LIN {X 0,Y 567.172,Z 389.799,A -85,B 0,C 180,E1 24706.932,E2 24706.932} C_VEL
LIN {X 0,Y 570.884,Z 340.567,A -85,B 0,C 180,E1 24705.981,E2 24705.981} C_VEL
LIN {X 0,Y 571.881,Z 338.159,A -85,B 0,C 180,E1 24705.833,E2 24705.833} C_VEL
LIN {X 0,Y 579.094,Z 319.344,A -85,B 0,C 180,E1 24704.229,E2 24704.229} C_VEL
LIN {X 0,Y 582.937,Z 311.16,A -85,B 0,C 180,E1 24703.458,E2 24703.458} C_VEL
LIN {X 0,Y 582.832,Z 309.162,A -85,B 0,C 180,E1 24702.394,E2 24702.394} C_VEL
LIN {X 0,Y 582.89,Z 308.585,A -85,B 0,C 180,E1 24701.727,E2 24701.727} C_VEL
LIN {X 0,Y 582.338,Z 310.355,A -85,B 0,C 180,E1 24700.405,E2 24700.405} C_VEL
LIN {X 0,Y 574.337,Z 326.452,A -85,B 0,C 180,E1 24698.682,E2 24698.682} C_VEL
LIN {X 0,Y 566.735,Z 346.819,A -85,B 0,C 180,E1 24696.671,E2 24696.671} C_VEL
LIN {X 0,Y 559.494,Z 373.809,A -85,B 0,C 180,E1 24694.198,E2 24694.198} C_VEL
LIN {X 0,Y 554.301,Z 400.115,A -85,B 0,C 180,E1 24691.96,E2 24691.96} C_VEL
LIN {X 0,Y 555.519,Z 423.333,A -85,B 0,C 180,E1 24690.693,E2 24690.693} C_VEL
LIN {X 0,Y 556.922,Z 451.305,A -85,B 0,C 180,E1 24689.365,E2 24689.365} C_VEL
LIN {X 0,Y 558.184,Z 484.283,A -85,B 0,C 180,E1 24688.02,E2 24688.02} C_VEL
LIN {X 0,Y 558.47,Z 501.799,A -85,B 0,C 180,E1 24687.4,E2 24687.4} C_VEL
LIN {X 0,Y 549.884,Z 603.402,A -85,B 0,C 180,E1 24685.067,E2 24685.067} C_VEL
LIN {X 0,Y 544.198,Z 689.935,A -85,B 0,C 180,E1 24683.104,E2 24683.104} C_VEL
LIN {X 0,Y 542.555,Z 713.994,A -85,B 0,C 180,E1 24682.34,E2 24682.34} C_VEL
LIN {X 0,Y 541.005,Z 736.005,A -85,B 0,C 180,E1 24681.432,E2 24681.432} C_VEL
LIN {X 0,Y 539.398,Z 756.989,A -85,B 0,C 180,E1 24680.339,E2 24680.339} C_VEL
LIN {X 0,Y 538.011,Z 774.87,A -85,B 0,C 180,E1 24679.205,E2 24679.205} C_VEL
LIN {X 0,Y 536.611,Z 791.893,A -85,B 0,C 180,E1 24677.906,E2 24677.906} C_VEL
LIN {X 0,Y 535.34,Z 806.843,A -85,B 0,C 180,E1 24676.549,E2 24676.549} C_VEL
LIN {X 0,Y 534.145,Z 820.367,A -85,B 0,C 180,E1 24675.082,E2 24675.082} C_VEL
LIN {X 0,Y 533.023,Z 832.916,A -85,B 0,C 180,E1 24673.451,E2 24673.451} C_VEL
LIN {X 0,Y 532.018,Z 843.847,A -85,B 0,C 180,E1 24671.711,E2 24671.711} C_VEL
LIN {X 0,Y 531.163,Z 853.18,A -85,B 0,C 180,E1 24669.864,E2 24669.864} C_VEL
LIN {X 0,Y 530.507,Z 860.457,A -85,B 0,C 180,E1 24668.017,E2 24668.017} C_VEL
LIN {X 0,Y 530,Z 866.128,A -85,B 0,C 180,E1 24666.065,E2 24666.065} C_VEL
LIN {X 0,Y 529.624,Z 869.937,A -85,B 0,C 180,E1 24664.114,E2 24664.114} C_VEL
LIN {X 0,Y 529.372,Z 871.943,A -85,B 0,C 180,E1 24662.165,E2 24662.165} C_VEL
LIN {X 0,Y 529.209,Z 872.179,A -85,B 0,C 180,E1 24660.108,E2 24660.108} C_VEL
LIN {X 0,Y 529.126,Z 870.512,A -85,B 0,C 180,E1 24658.051,E2 24658.051} C_VEL
LIN {X 0,Y 529.146,Z 867.199,A -85,B 0,C 180,E1 24656.099,E2 24656.099} C_VEL
LIN {X 0,Y 529.276,Z 862.125,A -85,B 0,C 180,E1 24654.145,E2 24654.145} C_VEL
LIN {X 0,Y 529.52,Z 855.186,A -85,B 0,C 180,E1 24652.186,E2 24652.186} C_VEL
LIN {X 0,Y 529.941,Z 846.185,A -85,B 0,C 180,E1 24650.223,E2 24650.223} C_VEL
LIN {X 0,Y 530.543,Z 835.567,A -85,B 0,C 180,E1 24648.366,E2 24648.366} C_VEL
LIN {X 0,Y 531.311,Z 823.375,A -85,B 0,C 180,E1 24646.616,E2 24646.616} C_VEL
LIN {X 0,Y 532.271,Z 809.122,A -85,B 0,C 180,E1 24644.921,E2 24644.921} C_VEL
LIN {X 0,Y 533.351,Z 793.597,A -85,B 0,C 180,E1 24643.387,E2 24643.387} C_VEL
LIN {X 0,Y 534.503,Z 776.998,A -85,B 0,C 180,E1 24642.021,E2 24642.021} C_VEL
LIN {X 0,Y 535.659,Z 759.422,A -85,B 0,C 180,E1 24640.82,E2 24640.82} C_VEL
LIN {X 0,Y 536.845,Z 740.956,A -85,B 0,C 180,E1 24639.788,E2 24639.788} C_VEL
LIN {X 0,Y 537.985,Z 720.972,A -85,B 0,C 180,E1 24638.894,E2 24638.894} C_VEL
LIN {X 0,Y 538.984,Z 700.182,A -85,B 0,C 180,E1 24638.188,E2 24638.188} C_VEL
LIN {X 0,Y 539.819,Z 679.295,A -85,B 0,C 180,E1 24637.684,E2 24637.684} C_VEL
LIN {X 0,Y 545.343,Z 494.327,A -85,B 0,C 180,E1 24634.546,E2 24634.546} C_VEL
LIN {X 0,Y 540.838,Z 450.424,A -85,B 0,C 180,E1 24633.456,E2 24633.456} C_VEL
LIN {X 0,Y 544.277,Z 398.054,A -85,B 0,C 180,E1 24629.86,E2 24629.86} C_VEL
LIN {X 0,Y 547.874,Z 348.579,A -85,B 0,C 180,E1 24626.428,E2 24626.428} C_VEL
LIN {X 0,Y 552.064,Z 296.542,A -85,B 0,C 180,E1 24622.776,E2 24622.776} C_VEL
LIN {X 0,Y 553.399,Z 279.163,A -85,B 0,C 180,E1 24621.532,E2 24621.532} C_VEL
LIN {X 0,Y 544.537,Z 255.5,A -85,B 0,C 180,E1 24618.998,E2 24618.998} C_VEL
LIN {X 0,Y 535.075,Z 232.411,A -85,B 0,C 180,E1 24616.318,E2 24616.318} C_VEL
LIN {X 0,Y 534.781,Z 231.7,A -85,B 0,C 180,E1 24616.227,E2 24616.227} C_VEL
LIN {X 0,Y 536.691,Z 232.864,A -85,B 0,C 180,E1 24615.941,E2 24615.941} C_VEL
LIN {X 0,Y 546.06,Z 252.219,A -85,B 0,C 180,E1 24613.597,E2 24613.597} C_VEL
LIN {X 0,Y 554.586,Z 272.537,A -85,B 0,C 180,E1 24611.251,E2 24611.251} C_VEL
LIN {X 0,Y 561.348,Z 291.078,A -85,B 0,C 180,E1 24609.21,E2 24609.21} C_VEL
LIN {X 0,Y 561.17,Z 298.745,A -85,B 0,C 180,E1 24608.658,E2 24608.658} C_VEL
LIN {X 0,Y 560.235,Z 305.401,A -85,B 0,C 180,E1 24608.261,E2 24608.261} C_VEL
LIN {X 0,Y 555.035,Z 324.312,A -85,B 0,C 180,E1 24607.416,E2 24607.416} C_VEL
LIN {X 0,Y 554.398,Z 330.093,A -85,B 0,C 180,E1 24607.081,E2 24607.081} C_VEL
LIN {X 0,Y 554.416,Z 348.963,A -85,B 0,C 180,E1 24605.852,E2 24605.852} C_VEL
LIN {X 0,Y 552.164,Z 359.982,A -85,B 0,C 180,E1 24605.442,E2 24605.442} C_VEL
LIN {X 0,Y 549.54,Z 449.417,A -85,B 0,C 180,E1 24604.138,E2 24604.138} C_VEL
LIN {X 0,Y 546.257,Z 527.382,A -85,B 0,C 180,E1 24602.815,E2 24602.815} C_VEL
LIN {X 0,Y 541.758,Z 616.567,A -85,B 0,C 180,E1 24601.087,E2 24601.087} C_VEL
LIN {X 0,Y 540.542,Z 646.224,A -85,B 0,C 180,E1 24600.4,E2 24600.4} C_VEL
LIN {X 0,Y 539.38,Z 668.071,A -85,B 0,C 180,E1 24599.698,E2 24599.698} C_VEL
LIN {X 0,Y 537.858,Z 689.945,A -85,B 0,C 180,E1 24598.783,E2 24598.783} C_VEL
LIN {X 0,Y 536.147,Z 710.107,A -85,B 0,C 180,E1 24597.73,E2 24597.73} C_VEL
LIN {X 0,Y 534.288,Z 729.488,A -85,B 0,C 180,E1 24596.509,E2 24596.509} C_VEL
LIN {X 0,Y 532.25,Z 748.721,A -85,B 0,C 180,E1 24595.064,E2 24595.064} C_VEL
LIN {X 0,Y 530.139,Z 767.337,A -85,B 0,C 180,E1 24593.403,E2 24593.403} C_VEL
LIN {X 0,Y 528.194,Z 784.001,A -85,B 0,C 180,E1 24591.645,E2 24591.645} C_VEL
LIN {X 0,Y 526.509,Z 798.406,A -85,B 0,C 180,E1 24589.873,E2 24589.873} C_VEL
LIN {X 0,Y 524.913,Z 812.343,A -85,B 0,C 180,E1 24587.86,E2 24587.86} C_VEL
LIN {X 0,Y 523.561,Z 824.713,A -85,B 0,C 180,E1 24585.732,E2 24585.732} C_VEL
LIN {X 0,Y 522.516,Z 835.264,A -85,B 0,C 180,E1 24583.562,E2 24583.562} C_VEL
LIN {X 0,Y 521.742,Z 844.408,A -85,B 0,C 180,E1 24581.273,E2 24581.273} C_VEL
LIN {X 0,Y 521.227,Z 851.534,A -85,B 0,C 180,E1 24579.051,E2 24579.051} C_VEL
LIN {X 0,Y 520.916,Z 857.237,A -85,B 0,C 180,E1 24576.724,E2 24576.724} C_VEL
LIN {X 0,Y 520.738,Z 861.151,A -85,B 0,C 180,E1 24574.405,E2 24574.405} C_VEL
LIN {X 0,Y 520.657,Z 863.456,A -85,B 0,C 180,E1 24572.091,E2 24572.091} C_VEL
LIN {X 0,Y 520.639,Z 864.185,A -85,B 0,C 180,E1 24569.78,E2 24569.78} C_VEL
LIN {X 0,Y 520.658,Z 863.243,A -85,B 0,C 180,E1 24567.468,E2 24567.468} C_VEL
LIN {X 0,Y 520.758,Z 860.648,A -85,B 0,C 180,E1 24565.154,E2 24565.154} C_VEL
LIN {X 0,Y 520.942,Z 856.196,A -85,B 0,C 180,E1 24562.722,E2 24562.722} C_VEL
LIN {X 0,Y 521.293,Z 850.544,A -85,B 0,C 180,E1 24560.505,E2 24560.505} C_VEL
LIN {X 0,Y 521.889,Z 842.757,A -85,B 0,C 180,E1 24558.17,E2 24558.17} C_VEL
LIN {X 0,Y 522.691,Z 833.442,A -85,B 0,C 180,E1 24555.94,E2 24555.94} C_VEL
LIN {X 0,Y 523.79,Z 822.558,A -85,B 0,C 180,E1 24553.783,E2 24553.783} C_VEL
LIN {X 0,Y 525.167,Z 809.983,A -85,B 0,C 180,E1 24551.69,E2 24551.69} C_VEL
LIN {X 0,Y 526.732,Z 796.54,A -85,B 0,C 180,E1 24549.788,E2 24549.788} C_VEL
LIN {X 0,Y 528.506,Z 781.567,A -85,B 0,C 180,E1 24547.979,E2 24547.979} C_VEL
LIN {X 0,Y 530.475,Z 764.694,A -85,B 0,C 180,E1 24546.247,E2 24546.247} C_VEL
LIN {X 0,Y 532.444,Z 747.087,A -85,B 0,C 180,E1 24544.708,E2 24544.708} C_VEL
LIN {X 0,Y 534.424,Z 728.325,A -85,B 0,C 180,E1 24543.318,E2 24543.318} C_VEL
LIN {X 0,Y 536.282,Z 708.692,A -85,B 0,C 180,E1 24542.096,E2 24542.096} C_VEL
LIN {X 0,Y 537.972,Z 688.594,A -85,B 0,C 180,E1 24541.062,E2 24541.062} C_VEL
LIN {X 0,Y 539.445,Z 667.47,A -85,B 0,C 180,E1 24540.185,E2 24540.185} C_VEL
LIN {X 0,Y 540.613,Z 645.234,A -85,B 0,C 180,E1 24539.477,E2 24539.477} C_VEL
LIN {X 0,Y 541.962,Z 612.731,A -85,B 0,C 180,E1 24538.738,E2 24538.738} C_VEL
LIN {X 0,Y 546.474,Z 523.52,A -85,B 0,C 180,E1 24537.02,E2 24537.02} C_VEL
LIN {X 0,Y 549.681,Z 446.416,A -85,B 0,C 180,E1 24535.721,E2 24535.721} C_VEL
LIN {X 0,Y 552.294,Z 358.711,A -85,B 0,C 180,E1 24534.437,E2 24534.437} C_VEL
LIN {X 0,Y 554.559,Z 348.099,A -85,B 0,C 180,E1 24534,E2 24534} C_VEL
LIN {X 0,Y 554.663,Z 312.521,A -85,B 0,C 180,E1 24531.609,E2 24531.609} C_VEL
LIN {X 0,Y 554.973,Z 294.272,A -85,B 0,C 180,E1 24530.293,E2 24530.293} C_VEL
LIN {X 0,Y 547.767,Z 275.074,A -85,B 0,C 180,E1 24528.139,E2 24528.139} C_VEL
LIN {X 0,Y 539.853,Z 256.334,A -85,B 0,C 180,E1 24525.942,E2 24525.942} C_VEL
LIN {X 0,Y 532.349,Z 240.84,A -85,B 0,C 180,E1 24524.024,E2 24524.024} C_VEL
LIN {X 0,Y 526.336,Z 229.281,A -85,B 0,C 180,E1 24522.555,E2 24522.555} C_VEL
LIN {X 0,Y 523.694,Z 224.562,A -85,B 0,C 180,E1 24521.933,E2 24521.933} C_VEL
LIN {X 0,Y 521.964,Z 221.334,A -85,B 0,C 180,E1 24521.515,E2 24521.515} C_VEL
LIN {X 0,Y 521.744,Z 220.235,A -85,B 0,C 180,E1 24521.39,E2 24521.39} C_VEL
LIN {X 0,Y 521.743,Z 220.233,A -85,B 0,C 180,E1 24517.965,E2 24517.965} C_VEL
LIN {X 0,Y 521.737,Z 220.239,A -85,B 0,C 180,E1 24514.505,E2 24514.505} C_VEL
LIN {X 0,Y 521.735,Z 220.239,A -85,B 0,C 180,E1 24511.033,E2 24511.033} C_VEL
LIN {X 0,Y 521.739,Z 220.219,A -85,B 0,C 180,E1 24507.632,E2 24507.632} C_VEL
LIN {X 0,Y 521.742,Z 220.211,A -85,B 0,C 180,E1 24504.185,E2 24504.185} C_VEL
LIN {X 0,Y 521.737,Z 220.238,A -85,B 0,C 180,E1 24500.734,E2 24500.734} C_VEL
LIN {X 0,Y 521.741,Z 220.21,A -85,B 0,C 180,E1 24497.281,E2 24497.281} C_VEL
LIN {X 0,Y 521.732,Z 220.223,A -85,B 0,C 180,E1 24493.861,E2 24493.861} C_VEL
LIN {X 0,Y 521.742,Z 220.225,A -85,B 0,C 180,E1 24490.378,E2 24490.378} C_VEL
LIN {X 0,Y 521.745,Z 220.21,A -85,B 0,C 180,E1 24486.922,E2 24486.922} C_VEL
LIN {X 0,Y 521.729,Z 220.239,A -85,B 0,C 180,E1 24483.406,E2 24483.406} C_VEL
LIN {X 0,Y 521.726,Z 220.202,A -85,B 0,C 180,E1 24479.89,E2 24479.89} C_VEL
LIN {X 0,Y 521.744,Z 220.238,A -85,B 0,C 180,E1 24476.484,E2 24476.484} C_VEL
LIN {X 0,Y 521.744,Z 220.198,A -85,B 0,C 180,E1 24472.955,E2 24472.955} C_VEL
LIN {X 0,Y 521.72,Z 220.241,A -85,B 0,C 180,E1 24469.476,E2 24469.476} C_VEL
LIN {X 0,Y 521.739,Z 220.242,A -85,B 0,C 180,E1 24466.026,E2 24466.026} C_VEL
LIN {X 0,Y 521.749,Z 220.241,A -85,B 0,C 180,E1 24462.605,E2 24462.605} C_VEL
LIN {X 0,Y 521.717,Z 220.239,A -85,B 0,C 180,E1 24459.233,E2 24459.233} C_VEL
LIN {X 0,Y 521.722,Z 220.235,A -85,B 0,C 180,E1 24455.787,E2 24455.787} C_VEL
LIN {X 0,Y 521.753,Z 220.235,A -85,B 0,C 180,E1 24452.369,E2 24452.369} C_VEL
LIN {X 0,Y 521.722,Z 220.239,A -85,B 0,C 180,E1 24448.946,E2 24448.946} C_VEL
LIN {X 0,Y 521.754,Z 220.325,A -85,B 0,C 180,E1 24446.612,E2 24446.612} C_VEL
LIN {X 0,Y 522.874,Z 223.439,A -85,B 0,C 180,E1 24446.187,E2 24446.187} C_VEL
LIN {X 0,Y 524.045,Z 225.27,A -85,B 0,C 180,E1 24445.878,E2 24445.878} C_VEL
LIN {X 0,Y 525.794,Z 228.852,A -85,B 0,C 180,E1 24445.347,E2 24445.347} C_VEL
LIN {X 0,Y 533.823,Z 244.524,A -85,B 0,C 180,E1 24443.04,E2 24443.04} C_VEL
LIN {X 0,Y 543.759,Z 264.219,A -85,B 0,C 180,E1 24440.351,E2 24440.351} C_VEL
LIN {X 0,Y 556.286,Z 289.963,A -85,B 0,C 180,E1 24437.168,E2 24437.168} C_VEL
LIN {X 0,Y 561.303,Z 300.628,A -85,B 0,C 180,E1 24435.946,E2 24435.946} C_VEL
LIN {X 0,Y 559.967,Z 313.808,A -85,B 0,C 180,E1 24435.173,E2 24435.173} C_VEL
LIN {X 0,Y 562.81,Z 340.382,A -85,B 0,C 180,E1 24434.457,E2 24434.457} C_VEL
LIN {X 0,Y 554.944,Z 572.433,A -85,B 0,C 180,E1 24430.918,E2 24430.918} C_VEL
LIN {X 0,Y 551.384,Z 692.781,A -85,B 0,C 180,E1 24429.119,E2 24429.119} C_VEL
LIN {X 0,Y 549.935,Z 717.309,A -85,B 0,C 180,E1 24428.579,E2 24428.579} C_VEL
LIN {X 0,Y 548.22,Z 740.807,A -85,B 0,C 180,E1 24427.893,E2 24427.893} C_VEL
LIN {X 0,Y 546.127,Z 763.625,A -85,B 0,C 180,E1 24427.035,E2 24427.035} C_VEL
LIN {X 0,Y 543.758,Z 786.648,A -85,B 0,C 180,E1 24425.992,E2 24425.992} C_VEL
LIN {X 0,Y 541.136,Z 809.081,A -85,B 0,C 180,E1 24424.753,E2 24424.753} C_VEL
LIN {X 0,Y 538.432,Z 830.883,A -85,B 0,C 180,E1 24423.345,E2 24423.345} C_VEL
LIN {X 0,Y 535.859,Z 850.246,A -85,B 0,C 180,E1 24421.875,E2 24421.875} C_VEL
LIN {X 0,Y 533.106,Z 870.475,A -85,B 0,C 180,E1 24420.114,E2 24420.114} C_VEL
LIN {X 0,Y 530.656,Z 888,A -85,B 0,C 180,E1 24418.348,E2 24418.348} C_VEL
LIN {X 0,Y 528.37,Z 904.978,A -85,B 0,C 180,E1 24416.405,E2 24416.405} C_VEL
LIN {X 0,Y 526.295,Z 920.525,A -85,B 0,C 180,E1 24414.348,E2 24414.348} C_VEL
LIN {X 0,Y 524.481,Z 935.456,A -85,B 0,C 180,E1 24412.099,E2 24412.099} C_VEL
LIN {X 0,Y 523.037,Z 948.215,A -85,B 0,C 180,E1 24409.854,E2 24409.854} C_VEL
LIN {X 0,Y 521.869,Z 960.375,A -85,B 0,C 180,E1 24407.391,E2 24407.391} C_VEL
LIN {X 0,Y 521.085,Z 970.191,A -85,B 0,C 180,E1 24405.013,E2 24405.013} C_VEL
LIN {X 0,Y 520.553,Z 978.856,A -85,B 0,C 180,E1 24402.536,E2 24402.536} C_VEL
LIN {X 0,Y 520.257,Z 985.967,A -85,B 0,C 180,E1 24399.961,E2 24399.961} C_VEL
LIN {X 0,Y 520.116,Z 990.812,A -85,B 0,C 180,E1 24397.734,E2 24397.734} C_VEL
LIN {X 0,Y 520.085,Z 994.867,A -85,B 0,C 180,E1 24395.184,E2 24395.184} C_VEL
LIN {X 0,Y 520.101,Z 997.064,A -85,B 0,C 180,E1 24392.865,E2 24392.865} C_VEL
LIN {X 0,Y 520.12,Z 997.946,A -85,B 0,C 180,E1 24390.771,E2 24390.771} C_VEL
LIN {X 0,Y 520.139,Z 997.696,A -85,B 0,C 180,E1 24388.439,E2 24388.439} C_VEL
LIN {X 0,Y 520.139,Z 995.709,A -85,B 0,C 180,E1 24385.811,E2 24385.811} C_VEL
LIN {X 0,Y 520.149,Z 992.525,A -85,B 0,C 180,E1 24383.488,E2 24383.488} C_VEL
LIN {X 0,Y 520.233,Z 987.22,A -85,B 0,C 180,E1 24380.82,E2 24380.82} C_VEL
LIN {X 0,Y 520.439,Z 980.92,A -85,B 0,C 180,E1 24378.474,E2 24378.474} C_VEL
LIN {X 0,Y 520.81,Z 973.556,A -85,B 0,C 180,E1 24376.228,E2 24376.228} C_VEL
LIN {X 0,Y 521.5,Z 963.155,A -85,B 0,C 180,E1 24373.629,E2 24373.629} C_VEL
LIN {X 0,Y 522.274,Z 953.521,A -85,B 0,C 180,E1 24371.585,E2 24371.585} C_VEL
LIN {X 0,Y 523.524,Z 940.476,A -85,B 0,C 180,E1 24369.191,E2 24369.191} C_VEL
LIN {X 0,Y 524.882,Z 927.409,A -85,B 0,C 180,E1 24367.131,E2 24367.131} C_VEL
LIN {X 0,Y 526.69,Z 911.753,A -85,B 0,C 180,E1 24364.953,E2 24364.953} C_VEL
LIN {X 0,Y 528.751,Z 894.474,A -85,B 0,C 180,E1 24362.887,E2 24362.887} C_VEL
LIN {X 0,Y 531.057,Z 875.875,A -85,B 0,C 180,E1 24360.937,E2 24360.937} C_VEL
LIN {X 0,Y 533.395,Z 856.932,A -85,B 0,C 180,E1 24359.219,E2 24359.219} C_VEL
LIN {X 0,Y 536.068,Z 835.167,A -85,B 0,C 180,E1 24357.508,E2 24357.508} C_VEL
LIN {X 0,Y 538.313,Z 815.895,A -85,B 0,C 180,E1 24356.199,E2 24356.199} C_VEL
LIN {X 0,Y 540.838,Z 792.483,A -85,B 0,C 180,E1 24354.838,E2 24354.838} C_VEL
LIN {X 0,Y 543.143,Z 769.878,A -85,B 0,C 180,E1 24353.739,E2 24353.739} C_VEL
LIN {X 0,Y 545.171,Z 746.679,A -85,B 0,C 180,E1 24352.819,E2 24352.819} C_VEL
LIN {X 0,Y 546.946,Z 723.653,A -85,B 0,C 180,E1 24352.081,E2 24352.081} C_VEL
LIN {X 0,Y 548.337,Z 699.785,A -85,B 0,C 180,E1 24351.51,E2 24351.51} C_VEL
LIN {X 0,Y 549.321,Z 674.5,A -85,B 0,C 180,E1 24351.074,E2 24351.074} C_VEL
LIN {X 0,Y 552.201,Z 576.067,A -85,B 0,C 180,E1 24349.588,E2 24349.588} C_VEL
LIN {X 0,Y 556.018,Z 486.791,A -85,B 0,C 180,E1 24348.088,E2 24348.088} C_VEL
LIN {X 0,Y 561.161,Z 403.595,A -85,B 0,C 180,E1 24346.558,E2 24346.558} C_VEL
LIN {X 0,Y 566.111,Z 343.623,A -85,B 0,C 180,E1 24345.37,E2 24345.37} C_VEL
LIN {X 0,Y 567.547,Z 340.563,A -85,B 0,C 180,E1 24345.194,E2 24345.194} C_VEL
LIN {X 0,Y 575.021,Z 323.124,A -85,B 0,C 180,E1 24343.657,E2 24343.657} C_VEL
LIN {X 0,Y 578.257,Z 316.88,A -85,B 0,C 180,E1 24343.066,E2 24343.066} C_VEL
LIN {X 0,Y 578.346,Z 315.09,A -85,B 0,C 180,E1 24341.828,E2 24341.828} C_VEL
LIN {X 0,Y 577.731,Z 316.371,A -85,B 0,C 180,E1 24340.762,E2 24340.762} C_VEL
LIN {X 0,Y 568.969,Z 332.766,A -85,B 0,C 180,E1 24338.987,E2 24338.987} C_VEL
LIN {X 0,Y 561.23,Z 352.221,A -85,B 0,C 180,E1 24337.027,E2 24337.027} C_VEL
LIN {X 0,Y 553.999,Z 376.806,A -85,B 0,C 180,E1 24334.711,E2 24334.711} C_VEL
LIN {X 0,Y 549.797,Z 396.074,A -85,B 0,C 180,E1 24333.028,E2 24333.028} C_VEL
LIN {X 0,Y 550.632,Z 420.862,A -85,B 0,C 180,E1 24331.577,E2 24331.577} C_VEL
LIN {X 0,Y 551.732,Z 450.81,A -85,B 0,C 180,E1 24330.08,E2 24330.08} C_VEL
LIN {X 0,Y 552.582,Z 483.66,A -85,B 0,C 180,E1 24328.683,E2 24328.683} C_VEL
LIN {X 0,Y 552.788,Z 503.004,A -85,B 0,C 180,E1 24327.969,E2 24327.969} C_VEL
LIN {X 0,Y 543.196,Z 609.107,A -85,B 0,C 180,E1 24325.463,E2 24325.463} C_VEL
LIN {X 0,Y 537.537,Z 689.387,A -85,B 0,C 180,E1 24323.586,E2 24323.586} C_VEL
LIN {X 0,Y 535.83,Z 712.83,A -85,B 0,C 180,E1 24322.839,E2 24322.839} C_VEL
LIN {X 0,Y 534.14,Z 734.712,A -85,B 0,C 180,E1 24321.929,E2 24321.929} C_VEL
LIN {X 0,Y 532.54,Z 754.757,A -85,B 0,C 180,E1 24320.9,E2 24320.9} C_VEL
LIN {X 0,Y 530.937,Z 773.824,A -85,B 0,C 180,E1 24319.701,E2 24319.701} C_VEL
LIN {X 0,Y 529.443,Z 791.217,A -85,B 0,C 180,E1 24318.385,E2 24318.385} C_VEL
LIN {X 0,Y 527.95,Z 807.44,A -85,B 0,C 180,E1 24316.901,E2 24316.901} C_VEL
LIN {X 0,Y 526.676,Z 821.085,A -85,B 0,C 180,E1 24315.414,E2 24315.414} C_VEL
LIN {X 0,Y 525.456,Z 833.65,A -85,B 0,C 180,E1 24313.76,E2 24313.76} C_VEL
LIN {X 0,Y 524.372,Z 844.771,A -85,B 0,C 180,E1 24311.983,E2 24311.983} C_VEL
LIN {X 0,Y 523.445,Z 854.084,A -85,B 0,C 180,E1 24310.122,E2 24310.122} C_VEL
LIN {X 0,Y 522.727,Z 861.417,A -85,B 0,C 180,E1 24308.248,E2 24308.248} C_VEL
LIN {X 0,Y 522.168,Z 867.158,A -85,B 0,C 180,E1 24306.266,E2 24306.266} C_VEL
LIN {X 0,Y 521.752,Z 870.983,A -85,B 0,C 180,E1 24304.286,E2 24304.286} C_VEL
LIN {X 0,Y 521.458,Z 873.086,A -85,B 0,C 180,E1 24302.198,E2 24302.198} C_VEL
LIN {X 0,Y 521.288,Z 873.282,A -85,B 0,C 180,E1 24300.22,E2 24300.22} C_VEL
LIN {X 0,Y 521.191,Z 871.638,A -85,B 0,C 180,E1 24298.131,E2 24298.131} C_VEL
LIN {X 0,Y 521.209,Z 868.088,A -85,B 0,C 180,E1 24296.04,E2 24296.04} C_VEL
LIN {X 0,Y 521.345,Z 862.924,A -85,B 0,C 180,E1 24294.055,E2 24294.055} C_VEL
LIN {X 0,Y 521.604,Z 855.883,A -85,B 0,C 180,E1 24292.067,E2 24292.067} C_VEL
LIN {X 0,Y 522.02,Z 847.345,A -85,B 0,C 180,E1 24290.185,E2 24290.185} C_VEL
LIN {X 0,Y 522.64,Z 836.731,A -85,B 0,C 180,E1 24288.3,E2 24288.3} C_VEL
LIN {X 0,Y 523.432,Z 824.547,A -85,B 0,C 180,E1 24286.523,E2 24286.523} C_VEL
LIN {X 0,Y 524.389,Z 810.796,A -85,B 0,C 180,E1 24284.857,E2 24284.857} C_VEL
LIN {X 0,Y 525.493,Z 795.428,A -85,B 0,C 180,E1 24283.302,E2 24283.302} C_VEL
LIN {X 0,Y 526.724,Z 778.299,A -85,B 0,C 180,E1 24281.861,E2 24281.861} C_VEL
LIN {X 0,Y 527.917,Z 760.842,A -85,B 0,C 180,E1 24280.643,E2 24280.643} C_VEL
LIN {X 0,Y 529.12,Z 742.725,A -85,B 0,C 180,E1 24279.604,E2 24279.604} C_VEL
LIN {X 0,Y 530.265,Z 723.546,A -85,B 0,C 180,E1 24278.716,E2 24278.716} C_VEL
LIN {X 0,Y 531.332,Z 702.865,A -85,B 0,C 180,E1 24277.974,E2 24277.974} C_VEL
LIN {X 0,Y 532.259,Z 681.478,A -85,B 0,C 180,E1 24277.426,E2 24277.426} C_VEL
LIN {X 0,Y 538.097,Z 495.341,A -85,B 0,C 180,E1 24274.201,E2 24274.201} C_VEL
LIN {X 0,Y 533.475,Z 449.88,A -85,B 0,C 180,E1 24273.059,E2 24273.059} C_VEL
LIN {X 0,Y 537.156,Z 396.261,A -85,B 0,C 180,E1 24269.333,E2 24269.333} C_VEL
LIN {X 0,Y 540.798,Z 348.675,A -85,B 0,C 180,E1 24265.993,E2 24265.993} C_VEL
LIN {X 0,Y 545.201,Z 296.528,A -85,B 0,C 180,E1 24262.292,E2 24262.292} C_VEL
LIN {X 0,Y 546.276,Z 282.025,A -85,B 0,C 180,E1 24261.237,E2 24261.237} C_VEL
LIN {X 0,Y 537.787,Z 259.311,A -85,B 0,C 180,E1 24258.771,E2 24258.771} C_VEL
LIN {X 0,Y 529.445,Z 238.662,A -85,B 0,C 180,E1 24256.341,E2 24256.341} C_VEL
LIN {X 0,Y 531.632,Z 239.348,A -85,B 0,C 180,E1 24256.051,E2 24256.051} C_VEL
LIN {X 0,Y 539.955,Z 256.58,A -85,B 0,C 180,E1 24253.916,E2 24253.916} C_VEL
LIN {X 0,Y 547.54,Z 274.698,A -85,B 0,C 180,E1 24251.801,E2 24251.801} C_VEL
LIN {X 0,Y 554.992,Z 294.722,A -85,B 0,C 180,E1 24249.559,E2 24249.559} C_VEL
LIN {X 0,Y 554.398,Z 330.093,A -85,B 0,C 180,E1 24247.081,E2 24247.081} C_VEL
LIN {X 0,Y 553.581,Z 335.341,A -85,B 0,C 180,E1 24246.81,E2 24246.81} C_VEL
LIN {X 0,Y 547.836,Z 351.92,A -85,B 0,C 180,E1 24246.299,E2 24246.299} C_VEL
LIN {X 0,Y 545.655,Z 362.546,A -85,B 0,C 180,E1 24245.903,E2 24245.903} C_VEL
LIN {X 0,Y 542.944,Z 451.442,A -85,B 0,C 180,E1 24244.595,E2 24244.595} C_VEL
LIN {X 0,Y 539.626,Z 527.403,A -85,B 0,C 180,E1 24243.289,E2 24243.289} C_VEL
LIN {X 0,Y 535.005,Z 615.09,A -85,B 0,C 180,E1 24241.566,E2 24241.566} C_VEL
LIN {X 0,Y 533.624,Z 647.175,A -85,B 0,C 180,E1 24240.817,E2 24240.817} C_VEL
LIN {X 0,Y 532.402,Z 669.345,A -85,B 0,C 180,E1 24240.096,E2 24240.096} C_VEL
LIN {X 0,Y 530.865,Z 690.529,A -85,B 0,C 180,E1 24239.198,E2 24239.198} C_VEL
LIN {X 0,Y 529.086,Z 710.813,A -85,B 0,C 180,E1 24238.133,E2 24238.133} C_VEL
LIN {X 0,Y 527.153,Z 730.268,A -85,B 0,C 180,E1 24236.897,E2 24236.897} C_VEL
LIN {X 0,Y 525.02,Z 749.549,A -85,B 0,C 180,E1 24235.433,E2 24235.433} C_VEL
LIN {X 0,Y 522.942,Z 767.166,A -85,B 0,C 180,E1 24233.854,E2 24233.854} C_VEL
LIN {X 0,Y 521.033,Z 782.83,A -85,B 0,C 180,E1 24232.213,E2 24232.213} C_VEL
LIN {X 0,Y 519.068,Z 798.679,A -85,B 0,C 180,E1 24230.261,E2 24230.261} C_VEL
LIN {X 0,Y 517.376,Z 812.519,A -85,B 0,C 180,E1 24228.245,E2 24228.245} C_VEL
LIN {X 0,Y 515.997,Z 824.407,A -85,B 0,C 180,E1 24226.203,E2 24226.203} C_VEL
LIN {X 0,Y 514.817,Z 835.488,A -85,B 0,C 180,E1 24223.936,E2 24223.936} C_VEL
LIN {X 0,Y 513.987,Z 844.588,A -85,B 0,C 180,E1 24221.673,E2 24221.673} C_VEL
LIN {X 0,Y 513.4,Z 851.915,A -85,B 0,C 180,E1 24219.416,E2 24219.416} C_VEL
LIN {X 0,Y 513.02,Z 857.723,A -85,B 0,C 180,E1 24217.053,E2 24217.053} C_VEL
LIN {X 0,Y 512.827,Z 861.83,A -85,B 0,C 180,E1 24214.697,E2 24214.697} C_VEL
LIN {X 0,Y 512.724,Z 864.323,A -85,B 0,C 180,E1 24212.347,E2 24212.347} C_VEL
LIN {X 0,Y 512.715,Z 865.211,A -85,B 0,C 180,E1 24210,E2 24210} C_VEL
LIN {X 0,Y 512.721,Z 864.377,A -85,B 0,C 180,E1 24207.653,E2 24207.653} C_VEL
LIN {X 0,Y 512.823,Z 861.957,A -85,B 0,C 180,E1 24205.303,E2 24205.303} C_VEL
LIN {X 0,Y 513.013,Z 857.929,A -85,B 0,C 180,E1 24202.947,E2 24202.947} C_VEL
LIN {X 0,Y 513.376,Z 852.172,A -85,B 0,C 180,E1 24200.584,E2 24200.584} C_VEL
LIN {X 0,Y 513.959,Z 844.91,A -85,B 0,C 180,E1 24198.327,E2 24198.327} C_VEL
LIN {X 0,Y 514.778,Z 835.896,A -85,B 0,C 180,E1 24196.063,E2 24196.063} C_VEL
LIN {X 0,Y 515.881,Z 825.52,A -85,B 0,C 180,E1 24193.909,E2 24193.909} C_VEL
LIN {X 0,Y 517.236,Z 813.852,A -85,B 0,C 180,E1 24191.866,E2 24191.866} C_VEL
LIN {X 0,Y 518.962,Z 799.602,A -85,B 0,C 180,E1 24189.77,E2 24189.77} C_VEL
LIN {X 0,Y 520.817,Z 784.56,A -85,B 0,C 180,E1 24187.896,E2 24187.896} C_VEL
LIN {X 0,Y 522.772,Z 768.635,A -85,B 0,C 180,E1 24186.198,E2 24186.198} C_VEL
LIN {X 0,Y 524.953,Z 750.305,A -85,B 0,C 180,E1 24184.535,E2 24184.535} C_VEL
LIN {X 0,Y 527.06,Z 731.305,A -85,B 0,C 180,E1 24183.081,E2 24183.081} C_VEL
LIN {X 0,Y 528.977,Z 712.359,A -85,B 0,C 180,E1 24181.861,E2 24181.861} C_VEL
LIN {X 0,Y 530.751,Z 692.432,A -85,B 0,C 180,E1 24180.795,E2 24180.795} C_VEL
LIN {X 0,Y 532.312,Z 670.851,A -85,B 0,C 180,E1 24179.868,E2 24179.868} C_VEL
LIN {X 0,Y 533.516,Z 649.724,A -85,B 0,C 180,E1 24179.164,E2 24179.164} C_VEL
LIN {X 0,Y 534.659,Z 622.529,A -85,B 0,C 180,E1 24178.499,E2 24178.499} C_VEL
LIN {X 0,Y 539.133,Z 537.667,A -85,B 0,C 180,E1 24176.807,E2 24176.807} C_VEL
LIN {X 0,Y 542.511,Z 463.41,A -85,B 0,C 180,E1 24175.504,E2 24175.504} C_VEL
LIN {X 0,Y 544.936,Z 390.36,A -85,B 0,C 180,E1 24174.396,E2 24174.396} C_VEL
LIN {X 0,Y 545.777,Z 361.482,A -85,B 0,C 180,E1 24173.979,E2 24173.979} C_VEL
LIN {X 0,Y 548.279,Z 350.09,A -85,B 0,C 180,E1 24173.521,E2 24173.521} C_VEL
LIN {X 0,Y 548.418,Z 314.014,A -85,B 0,C 180,E1 24171.09,E2 24171.09} C_VEL
LIN {X 0,Y 548.648,Z 298.086,A -85,B 0,C 180,E1 24169.946,E2 24169.946} C_VEL
LIN {X 0,Y 541.116,Z 277.916,A -85,B 0,C 180,E1 24167.658,E2 24167.658} C_VEL
LIN {X 0,Y 533.24,Z 259.389,A -85,B 0,C 180,E1 24165.443,E2 24165.443} C_VEL
LIN {X 0,Y 524.905,Z 242.374,A -85,B 0,C 180,E1 24163.296,E2 24163.296} C_VEL
LIN {X 0,Y 518.482,Z 230.32,A -85,B 0,C 180,E1 24161.708,E2 24161.708} C_VEL
LIN {X 0,Y 515.867,Z 225.675,A -85,B 0,C 180,E1 24161.077,E2 24161.077} C_VEL
LIN {X 0,Y 514.115,Z 222.681,A -85,B 0,C 180,E1 24160.658,E2 24160.658} C_VEL
LIN {X 0,Y 513.798,Z 221.214,A -85,B 0,C 180,E1 24160.498,E2 24160.498} C_VEL
LIN {X 0,Y 513.791,Z 221.21,A -85,B 0,C 180,E1 24156.967,E2 24156.967} C_VEL
LIN {X 0,Y 513.805,Z 221.208,A -85,B 0,C 180,E1 24153.551,E2 24153.551} C_VEL
LIN {X 0,Y 513.805,Z 221.222,A -85,B 0,C 180,E1 24150.004,E2 24150.004} C_VEL
LIN {X 0,Y 513.798,Z 221.224,A -85,B 0,C 180,E1 24146.59,E2 24146.59} C_VEL
LIN {X 0,Y 513.8,Z 221.196,A -85,B 0,C 180,E1 24143.002,E2 24143.002} C_VEL
LIN {X 0,Y 513.797,Z 221.214,A -85,B 0,C 180,E1 24139.556,E2 24139.556} C_VEL
LIN {X 0,Y 513.8,Z 221.221,A -85,B 0,C 180,E1 24135.98,E2 24135.98} C_VEL
LIN {X 0,Y 513.797,Z 221.192,A -85,B 0,C 180,E1 24132.589,E2 24132.589} C_VEL
LIN {X 0,Y 513.806,Z 221.226,A -85,B 0,C 180,E1 24129.069,E2 24129.069} C_VEL
LIN {X 0,Y 513.785,Z 221.192,A -85,B 0,C 180,E1 24125.584,E2 24125.584} C_VEL
LIN {X 0,Y 513.802,Z 221.226,A -85,B 0,C 180,E1 24122.119,E2 24122.119} C_VEL
LIN {X 0,Y 513.802,Z 221.191,A -85,B 0,C 180,E1 24118.662,E2 24118.662} C_VEL
LIN {X 0,Y 513.795,Z 221.224,A -85,B 0,C 180,E1 24115.134,E2 24115.134} C_VEL
LIN {X 0,Y 513.78,Z 221.2,A -85,B 0,C 180,E1 24111.72,E2 24111.72} C_VEL
LIN {X 0,Y 513.808,Z 221.229,A -85,B 0,C 180,E1 24108.323,E2 24108.323} C_VEL
LIN {X 0,Y 513.812,Z 221.22,A -85,B 0,C 180,E1 24104.769,E2 24104.769} C_VEL
LIN {X 0,Y 513.779,Z 221.223,A -85,B 0,C 180,E1 24101.27,E2 24101.27} C_VEL
LIN {X 0,Y 513.779,Z 221.231,A -85,B 0,C 180,E1 24097.697,E2 24097.697} C_VEL
LIN {X 0,Y 513.812,Z 221.231,A -85,B 0,C 180,E1 24094.28,E2 24094.28} C_VEL
LIN {X 0,Y 513.801,Z 221.221,A -85,B 0,C 180,E1 24090.76,E2 24090.76} C_VEL
LIN {X 0,Y 513.781,Z 221.313,A -85,B 0,C 180,E1 24087.544,E2 24087.544} C_VEL
LIN {X 0,Y 515.013,Z 224.619,A -85,B 0,C 180,E1 24087.07,E2 24087.07} C_VEL
LIN {X 0,Y 516.201,Z 226.326,A -85,B 0,C 180,E1 24086.758,E2 24086.758} C_VEL
LIN {X 0,Y 525.585,Z 244.911,A -85,B 0,C 180,E1 24083.953,E2 24083.953} C_VEL
LIN {X 0,Y 535.655,Z 264.841,A -85,B 0,C 180,E1 24081.156,E2 24081.156} C_VEL
LIN {X 0,Y 547.492,Z 289.167,A -85,B 0,C 180,E1 24078.054,E2 24078.054} C_VEL
LIN {X 0,Y 554.609,Z 304.613,A -85,B 0,C 180,E1 24076.261,E2 24076.261} C_VEL
LIN {X 0,Y 553.588,Z 314.57,A -85,B 0,C 180,E1 24075.679,E2 24075.679} C_VEL
LIN {X 0,Y 556.414,Z 341.608,A -85,B 0,C 180,E1 24074.938,E2 24074.938} C_VEL
LIN {X 0,Y 547.903,Z 580.869,A -85,B 0,C 180,E1 24071.235,E2 24071.235} C_VEL
LIN {X 0,Y 544.443,Z 692.816,A -85,B 0,C 180,E1 24069.536,E2 24069.536} C_VEL
LIN {X 0,Y 542.93,Z 717.515,A -85,B 0,C 180,E1 24068.984,E2 24068.984} C_VEL
LIN {X 0,Y 541.124,Z 741.364,A -85,B 0,C 180,E1 24068.278,E2 24068.278} C_VEL
LIN {X 0,Y 538.988,Z 763.83,A -85,B 0,C 180,E1 24067.419,E2 24067.419} C_VEL
LIN {X 0,Y 536.611,Z 786.263,A -85,B 0,C 180,E1 24066.393,E2 24066.393} C_VEL
LIN {X 0,Y 533.939,Z 808.357,A -85,B 0,C 180,E1 24065.159,E2 24065.159} C_VEL
LIN {X 0,Y 531.121,Z 830.193,A -85,B 0,C 180,E1 24063.736,E2 24063.736} C_VEL
LIN {X 0,Y 528.363,Z 850.31,A -85,B 0,C 180,E1 24062.191,E2 24062.191} C_VEL
LIN {X 0,Y 525.519,Z 870.526,A -85,B 0,C 180,E1 24060.405,E2 24060.405} C_VEL
LIN {X 0,Y 523.04,Z 887.566,A -85,B 0,C 180,E1 24058.661,E2 24058.661} C_VEL
LIN {X 0,Y 520.548,Z 905.348,A -85,B 0,C 180,E1 24056.587,E2 24056.587} C_VEL
LIN {X 0,Y 518.526,Z 920.04,A -85,B 0,C 180,E1 24054.615,E2 24054.615} C_VEL
LIN {X 0,Y 516.62,Z 935.081,A -85,B 0,C 180,E1 24052.309,E2 24052.309} C_VEL
LIN {X 0,Y 515.125,Z 947.805,A -85,B 0,C 180,E1 24050.036,E2 24050.036} C_VEL
LIN {X 0,Y 513.93,Z 959.862,A -85,B 0,C 180,E1 24047.552,E2 24047.552} C_VEL
LIN {X 0,Y 513.116,Z 969.651,A -85,B 0,C 180,E1 24045.137,E2 24045.137} C_VEL
LIN {X 0,Y 512.574,Z 978.291,A -85,B 0,C 180,E1 24042.62,E2 24042.62} C_VEL
LIN {X 0,Y 512.276,Z 985.347,A -85,B 0,C 180,E1 24040.004,E2 24040.004} C_VEL
LIN {X 0,Y 512.135,Z 990.375,A -85,B 0,C 180,E1 24037.629,E2 24037.629} C_VEL
LIN {X 0,Y 512.127,Z 994.251,A -85,B 0,C 180,E1 24035.04,E2 24035.04} C_VEL
LIN {X 0,Y 512.146,Z 996.271,A -85,B 0,C 180,E1 24032.798,E2 24032.798} C_VEL
LIN {X 0,Y 512.166,Z 997.098,A -85,B 0,C 180,E1 24030.671,E2 24030.671} C_VEL
LIN {X 0,Y 512.187,Z 996.701,A -85,B 0,C 180,E1 24028.098,E2 24028.098} C_VEL
LIN {X 0,Y 512.182,Z 994.664,A -85,B 0,C 180,E1 24025.633,E2 24025.633} C_VEL
LIN {X 0,Y 512.19,Z 991.585,A -85,B 0,C 180,E1 24023.386,E2 24023.386} C_VEL
LIN {X 0,Y 512.276,Z 986.225,A -85,B 0,C 180,E1 24020.677,E2 24020.677} C_VEL
LIN {X 0,Y 512.482,Z 979.874,A -85,B 0,C 180,E1 24018.293,E2 24018.293} C_VEL
LIN {X 0,Y 512.885,Z 972.073,A -85,B 0,C 180,E1 24015.895,E2 24015.895} C_VEL
LIN {X 0,Y 513.582,Z 961.984,A -85,B 0,C 180,E1 24013.37,E2 24013.37} C_VEL
LIN {X 0,Y 514.442,Z 951.733,A -85,B 0,C 180,E1 24011.177,E2 24011.177} C_VEL
LIN {X 0,Y 515.831,Z 937.766,A -85,B 0,C 180,E1 24008.628,E2 24008.628} C_VEL
LIN {X 0,Y 517.342,Z 924.51,A -85,B 0,C 180,E1 24006.538,E2 24006.538} C_VEL
LIN {X 0,Y 519.377,Z 907.516,A -85,B 0,C 180,E1 24004.209,E2 24004.209} C_VEL
LIN {X 0,Y 521.504,Z 890.928,A -85,B 0,C 180,E1 24002.231,E2 24002.231} C_VEL
LIN {X 0,Y 523.962,Z 871.83,A -85,B 0,C 180,E1 24000.253,E2 24000.253} C_VEL
LIN {X 0,Y 526.505,Z 852.51,A -85,B 0,C 180,E1 23998.507,E2 23998.507} C_VEL
LIN {X 0,Y 529.134,Z 831.779,A -85,B 0,C 180,E1 23996.899,E2 23996.899} C_VEL
LIN {X 0,Y 531.627,Z 811.405,A -85,B 0,C 180,E1 23995.519,E2 23995.519} C_VEL
LIN {X 0,Y 534.108,Z 789.39,A -85,B 0,C 180,E1 23994.261,E2 23994.261} C_VEL
LIN {X 0,Y 536.515,Z 766.93,A -85,B 0,C 180,E1 23993.172,E2 23993.172} C_VEL
LIN {X 0,Y 538.617,Z 743.789,A -85,B 0,C 180,E1 23992.263,E2 23992.263} C_VEL
LIN {X 0,Y 540.513,Z 719.52,A -85,B 0,C 180,E1 23991.502,E2 23991.502} C_VEL
LIN {X 0,Y 541.892,Z 696.774,A -85,B 0,C 180,E1 23990.966,E2 23990.966} C_VEL
LIN {X 0,Y 543.2,Z 661.353,A -85,B 0,C 180,E1 23990.386,E2 23990.386} C_VEL
LIN {X 0,Y 546.299,Z 571.031,A -85,B 0,C 180,E1 23988.963,E2 23988.963} C_VEL
LIN {X 0,Y 550.506,Z 486.216,A -85,B 0,C 180,E1 23987.476,E2 23987.476} C_VEL
LIN {X 0,Y 555.962,Z 408.499,A -85,B 0,C 180,E1 23985.993,E2 23985.993} C_VEL
LIN {X 0,Y 561.718,Z 346.62,A -85,B 0,C 180,E1 23984.727,E2 23984.727} C_VEL
LIN {X 0,Y 563.414,Z 343.383,A -85,B 0,C 180,E1 23984.558,E2 23984.558} C_VEL
LIN {X 0,Y 571.56,Z 326.361,A -85,B 0,C 180,E1 23983.008,E2 23983.008} C_VEL
LIN {X 0,Y 573.618,Z 322.708,A -85,B 0,C 180,E1 23982.642,E2 23982.642} C_VEL
LIN {X 0,Y 573.653,Z 321.761,A -85,B 0,C 180,E1 23981.747,E2 23981.747} C_VEL
LIN {X 0,Y 573.256,Z 322.397,A -85,B 0,C 180,E1 23981.149,E2 23981.149} C_VEL
LIN {X 0,Y 564.185,Z 338.196,A -85,B 0,C 180,E1 23979.402,E2 23979.402} C_VEL
LIN {X 0,Y 555.357,Z 358.916,A -85,B 0,C 180,E1 23977.269,E2 23977.269} C_VEL
LIN {X 0,Y 548.201,Z 381.824,A -85,B 0,C 180,E1 23975.068,E2 23975.068} C_VEL
LIN {X 0,Y 545.95,Z 391.32,A -85,B 0,C 180,E1 23974.22,E2 23974.22} C_VEL
LIN {X 0,Y 546.136,Z 415.633,A -85,B 0,C 180,E1 23972.673,E2 23972.673} C_VEL
LIN {X 0,Y 546.636,Z 442.357,A -85,B 0,C 180,E1 23971.229,E2 23971.229} C_VEL
LIN {X 0,Y 547.093,Z 470.384,A -85,B 0,C 180,E1 23969.915,E2 23969.915} C_VEL
LIN {X 0,Y 547.38,Z 503.169,A -85,B 0,C 180,E1 23968.586,E2 23968.586} C_VEL
LIN {X 0,Y 536.921,Z 611.379,A -85,B 0,C 180,E1 23965.964,E2 23965.964} C_VEL
LIN {X 0,Y 530.828,Z 691.444,A -85,B 0,C 180,E1 23964.027,E2 23964.027} C_VEL
LIN {X 0,Y 529.01,Z 714.174,A -85,B 0,C 180,E1 23963.268,E2 23963.268} C_VEL
LIN {X 0,Y 527.139,Z 736.948,A -85,B 0,C 180,E1 23962.294,E2 23962.294} C_VEL
LIN {X 0,Y 525.344,Z 757.403,A -85,B 0,C 180,E1 23961.2,E2 23961.2} C_VEL
LIN {X 0,Y 523.665,Z 776.116,A -85,B 0,C 180,E1 23959.986,E2 23959.986} C_VEL
LIN {X 0,Y 521.997,Z 793.772,A -85,B 0,C 180,E1 23958.598,E2 23958.598} C_VEL
LIN {X 0,Y 520.492,Z 809.246,A -85,B 0,C 180,E1 23957.15,E2 23957.15} C_VEL
LIN {X 0,Y 519.102,Z 822.948,A -85,B 0,C 180,E1 23955.614,E2 23955.614} C_VEL
LIN {X 0,Y 517.844,Z 835.239,A -85,B 0,C 180,E1 23953.967,E2 23953.967} C_VEL
LIN {X 0,Y 516.683,Z 846.153,A -85,B 0,C 180,E1 23952.177,E2 23952.177} C_VEL
LIN {X 0,Y 515.749,Z 855.031,A -85,B 0,C 180,E1 23950.387,E2 23950.387} C_VEL
LIN {X 0,Y 514.958,Z 862.392,A -85,B 0,C 180,E1 23948.486,E2 23948.486} C_VEL
LIN {X 0,Y 514.341,Z 868.175,A -85,B 0,C 180,E1 23946.474,E2 23946.474} C_VEL
LIN {X 0,Y 513.885,Z 872.044,A -85,B 0,C 180,E1 23944.464,E2 23944.464} C_VEL
LIN {X 0,Y 513.568,Z 874.096,A -85,B 0,C 180,E1 23942.455,E2 23942.455} C_VEL
LIN {X 0,Y 513.371,Z 874.395,A -85,B 0,C 180,E1 23940.446,E2 23940.446} C_VEL
LIN {X 0,Y 513.263,Z 872.984,A -85,B 0,C 180,E1 23938.437,E2 23938.437} C_VEL
LIN {X 0,Y 513.257,Z 869.868,A -85,B 0,C 180,E1 23936.426,E2 23936.426} C_VEL
LIN {X 0,Y 513.365,Z 865.003,A -85,B 0,C 180,E1 23934.411,E2 23934.411} C_VEL
LIN {X 0,Y 513.607,Z 858.286,A -85,B 0,C 180,E1 23932.393,E2 23932.393} C_VEL
LIN {X 0,Y 514.03,Z 849.547,A -85,B 0,C 180,E1 23930.37,E2 23930.37} C_VEL
LIN {X 0,Y 514.645,Z 839.211,A -85,B 0,C 180,E1 23928.456,E2 23928.456} C_VEL
LIN {X 0,Y 515.438,Z 827.346,A -85,B 0,C 180,E1 23926.653,E2 23926.653} C_VEL
LIN {X 0,Y 516.435,Z 813.483,A -85,B 0,C 180,E1 23924.905,E2 23924.905} C_VEL
LIN {X 0,Y 517.549,Z 798.451,A -85,B 0,C 180,E1 23923.328,E2 23923.328} C_VEL
LIN {X 0,Y 518.745,Z 782.464,A -85,B 0,C 180,E1 23921.921,E2 23921.921} C_VEL
LIN {X 0,Y 519.999,Z 764.842,A -85,B 0,C 180,E1 23920.628,E2 23920.628} C_VEL
LIN {X 0,Y 521.266,Z 746.492,A -85,B 0,C 180,E1 23919.521,E2 23919.521} C_VEL
LIN {X 0,Y 522.517,Z 726.749,A -85,B 0,C 180,E1 23918.562,E2 23918.562} C_VEL
LIN {X 0,Y 523.668,Z 705.694,A -85,B 0,C 180,E1 23917.768,E2 23917.768} C_VEL
LIN {X 0,Y 524.648,Z 684.535,A -85,B 0,C 180,E1 23917.187,E2 23917.187} C_VEL
LIN {X 0,Y 526.783,Z 615.83,A -85,B 0,C 180,E1 23915.956,E2 23915.956} C_VEL
LIN {X 0,Y 530.822,Z 495.843,A -85,B 0,C 180,E1 23913.834,E2 23913.834} C_VEL
LIN {X 0,Y 526.163,Z 448.839,A -85,B 0,C 180,E1 23912.62,E2 23912.62} C_VEL
LIN {X 0,Y 530.122,Z 393.926,A -85,B 0,C 180,E1 23908.755,E2 23908.755} C_VEL
LIN {X 0,Y 533.885,Z 347.053,A -85,B 0,C 180,E1 23905.425,E2 23905.425} C_VEL
LIN {X 0,Y 538.606,Z 293.929,A -85,B 0,C 180,E1 23901.612,E2 23901.612} C_VEL
LIN {X 0,Y 539.286,Z 285.255,A -85,B 0,C 180,E1 23900.975,E2 23900.975} C_VEL
LIN {X 0,Y 530.654,Z 262.108,A -85,B 0,C 180,E1 23898.422,E2 23898.422} C_VEL
LIN {X 0,Y 524.046,Z 245.633,A -85,B 0,C 180,E1 23896.465,E2 23896.465} C_VEL
LIN {X 0,Y 525.887,Z 246.35,A -85,B 0,C 180,E1 23896.204,E2 23896.204} C_VEL
LIN {X 0,Y 526.934,Z 246.319,A -85,B 0,C 180,E1 23896.087,E2 23896.087} C_VEL
LIN {X 0,Y 535.312,Z 264.189,A -85,B 0,C 180,E1 23893.863,E2 23893.863} C_VEL
LIN {X 0,Y 543.501,Z 284.174,A -85,B 0,C 180,E1 23891.516,E2 23891.516} C_VEL
LIN {X 0,Y 548.692,Z 298.744,A -85,B 0,C 180,E1 23889.897,E2 23889.897} C_VEL
LIN {X 0,Y 548.114,Z 340.328,A -85,B 0,C 180,E1 23887.013,E2 23887.013} C_VEL
LIN {X 0,Y 548.17,Z 350.473,A -85,B 0,C 180,E1 23886.357,E2 23886.357} C_VEL
LIN {X 0,Y 547.836,Z 351.92,A -85,B 0,C 180,E1 23886.299,E2 23886.299} C_VEL
LIN {X 0,Y 545.728,Z 359.167,A -85,B 0,C 180,E1 23886.117,E2 23886.117} C_VEL
LIN {X 0,Y 541.701,Z 370.787,A -85,B 0,C 180,E1 23886.094,E2 23886.094} C_VEL
LIN {X 0,Y 539.162,Z 380.551,A -85,B 0,C 180,E1 23886.119,E2 23886.119} C_VEL
LIN {X 0,Y 538.574,Z 386.081,A -85,B 0,C 180,E1 23886.074,E2 23886.074} C_VEL
LIN {X 0,Y 536.112,Z 460.229,A -85,B 0,C 180,E1 23884.953,E2 23884.953} C_VEL
LIN {X 0,Y 532.615,Z 535.506,A -85,B 0,C 180,E1 23883.625,E2 23883.625} C_VEL
LIN {X 0,Y 527.969,Z 619.963,A -85,B 0,C 180,E1 23881.92,E2 23881.92} C_VEL
LIN {X 0,Y 526.652,Z 649.813,A -85,B 0,C 180,E1 23881.195,E2 23881.195} C_VEL
LIN {X 0,Y 525.398,Z 671.372,A -85,B 0,C 180,E1 23880.476,E2 23880.476} C_VEL
LIN {X 0,Y 523.721,Z 693.609,A -85,B 0,C 180,E1 23879.51,E2 23879.51} C_VEL
LIN {X 0,Y 521.795,Z 714.5,A -85,B 0,C 180,E1 23878.374,E2 23878.374} C_VEL
LIN {X 0,Y 519.775,Z 733.497,A -85,B 0,C 180,E1 23877.124,E2 23877.124} C_VEL
LIN {X 0,Y 517.656,Z 751.757,A -85,B 0,C 180,E1 23875.699,E2 23875.699} C_VEL
LIN {X 0,Y 515.416,Z 769.759,A -85,B 0,C 180,E1 23874.041,E2 23874.041} C_VEL
LIN {X 0,Y 513.35,Z 785.828,A -85,B 0,C 180,E1 23872.302,E2 23872.302} C_VEL
LIN {X 0,Y 511.482,Z 800.258,A -85,B 0,C 180,E1 23870.483,E2 23870.483} C_VEL
LIN {X 0,Y 509.605,Z 814.92,A -85,B 0,C 180,E1 23868.297,E2 23868.297} C_VEL
LIN {X 0,Y 508.104,Z 827.192,A -85,B 0,C 180,E1 23866.109,E2 23866.109} C_VEL
LIN {X 0,Y 506.952,Z 837.449,A -85,B 0,C 180,E1 23863.924,E2 23863.924} C_VEL
LIN {X 0,Y 506.087,Z 846.355,A -85,B 0,C 180,E1 23861.626,E2 23861.626} C_VEL
LIN {X 0,Y 505.478,Z 853.506,A -85,B 0,C 180,E1 23859.335,E2 23859.335} C_VEL
LIN {X 0,Y 505.1,Z 859.21,A -85,B 0,C 180,E1 23856.936,E2 23856.936} C_VEL
LIN {X 0,Y 504.891,Z 863.141,A -85,B 0,C 180,E1 23854.544,E2 23854.544} C_VEL
LIN {X 0,Y 504.788,Z 865.457,A -85,B 0,C 180,E1 23852.157,E2 23852.157} C_VEL
LIN {X 0,Y 504.765,Z 866.186,A -85,B 0,C 180,E1 23849.773,E2 23849.773} C_VEL
LIN {X 0,Y 504.792,Z 865.243,A -85,B 0,C 180,E1 23847.389,E2 23847.389} C_VEL
LIN {X 0,Y 504.912,Z 862.638,A -85,B 0,C 180,E1 23845.001,E2 23845.001} C_VEL
LIN {X 0,Y 505.142,Z 858.169,A -85,B 0,C 180,E1 23842.493,E2 23842.493} C_VEL
LIN {X 0,Y 505.561,Z 852.489,A -85,B 0,C 180,E1 23840.207,E2 23840.207} C_VEL
LIN {X 0,Y 506.247,Z 844.704,A -85,B 0,C 180,E1 23837.799,E2 23837.799} C_VEL
LIN {X 0,Y 507.204,Z 835.165,A -85,B 0,C 180,E1 23835.455,E2 23835.455} C_VEL
LIN {X 0,Y 508.42,Z 824.501,A -85,B 0,C 180,E1 23833.29,E2 23833.29} C_VEL
LIN {X 0,Y 509.982,Z 811.826,A -85,B 0,C 180,E1 23831.125,E2 23831.125} C_VEL
LIN {X 0,Y 511.731,Z 798.33,A -85,B 0,C 180,E1 23829.169,E2 23829.169} C_VEL
LIN {X 0,Y 513.696,Z 783.374,A -85,B 0,C 180,E1 23827.313,E2 23827.313} C_VEL
LIN {X 0,Y 515.928,Z 766.106,A -85,B 0,C 180,E1 23825.497,E2 23825.497} C_VEL
LIN {X 0,Y 518.212,Z 747.418,A -85,B 0,C 180,E1 23823.839,E2 23823.839} C_VEL
LIN {X 0,Y 520.39,Z 728.283,A -85,B 0,C 180,E1 23822.415,E2 23822.415} C_VEL
LIN {X 0,Y 522.309,Z 709.125,A -85,B 0,C 180,E1 23821.219,E2 23821.219} C_VEL
LIN {X 0,Y 524.169,Z 688.135,A -85,B 0,C 180,E1 23820.14,E2 23820.14} C_VEL
LIN {X 0,Y 525.754,Z 666.086,A -85,B 0,C 180,E1 23819.239,E2 23819.239} C_VEL
LIN {X 0,Y 526.902,Z 644.598,A -85,B 0,C 180,E1 23818.564,E2 23818.564} C_VEL
LIN {X 0,Y 528.98,Z 602.126,A -85,B 0,C 180,E1 23817.605,E2 23817.605} C_VEL
LIN {X 0,Y 533.44,Z 520.097,A -85,B 0,C 180,E1 23815.994,E2 23815.994} C_VEL
LIN {X 0,Y 536.587,Z 449.175,A -85,B 0,C 180,E1 23814.775,E2 23814.775} C_VEL
LIN {X 0,Y 539.419,Z 363.626,A -85,B 0,C 180,E1 23813.486,E2 23813.486} C_VEL
LIN {X 0,Y 542.032,Z 351.759,A -85,B 0,C 180,E1 23813.012,E2 23813.012} C_VEL
LIN {X 0,Y 542.205,Z 315.561,A -85,B 0,C 180,E1 23810.565,E2 23810.565} C_VEL
LIN {X 0,Y 542.378,Z 301.936,A -85,B 0,C 180,E1 23809.586,E2 23809.586} C_VEL
LIN {X 0,Y 535.091,Z 282.309,A -85,B 0,C 180,E1 23807.334,E2 23807.334} C_VEL
LIN {X 0,Y 527.023,Z 263.385,A -85,B 0,C 180,E1 23805.046,E2 23805.046} C_VEL
LIN {X 0,Y 518.207,Z 245.125,A -85,B 0,C 180,E1 23802.705,E2 23802.705} C_VEL
LIN {X 0,Y 510.724,Z 231.488,A -85,B 0,C 180,E1 23800.837,E2 23800.837} C_VEL
LIN {X 0,Y 508.165,Z 226.883,A -85,B 0,C 180,E1 23800.195,E2 23800.195} C_VEL
LIN {X 0,Y 506.179,Z 223.633,A -85,B 0,C 180,E1 23799.72,E2 23799.72} C_VEL
LIN {X 0,Y 505.871,Z 222.206,A -85,B 0,C 180,E1 23799.569,E2 23799.569} C_VEL
LIN {X 0,Y 505.864,Z 222.201,A -85,B 0,C 180,E1 23796.057,E2 23796.057} C_VEL
LIN {X 0,Y 505.859,Z 222.193,A -85,B 0,C 180,E1 23792.523,E2 23792.523} C_VEL
LIN {X 0,Y 505.857,Z 222.193,A -85,B 0,C 180,E1 23788.965,E2 23788.965} C_VEL
LIN {X 0,Y 505.868,Z 222.213,A -85,B 0,C 180,E1 23785.399,E2 23785.399} C_VEL
LIN {X 0,Y 505.859,Z 222.205,A -85,B 0,C 180,E1 23781.815,E2 23781.815} C_VEL
LIN {X 0,Y 505.862,Z 222.18,A -85,B 0,C 180,E1 23778.317,E2 23778.317} C_VEL
LIN {X 0,Y 505.864,Z 222.215,A -85,B 0,C 180,E1 23774.773,E2 23774.773} C_VEL
LIN {X 0,Y 505.858,Z 222.186,A -85,B 0,C 180,E1 23771.285,E2 23771.285} C_VEL
LIN {X 0,Y 505.851,Z 222.204,A -85,B 0,C 180,E1 23767.725,E2 23767.725} C_VEL
LIN {X 0,Y 505.861,Z 222.199,A -85,B 0,C 180,E1 23764.194,E2 23764.194} C_VEL
LIN {X 0,Y 505.864,Z 222.188,A -85,B 0,C 180,E1 23760.68,E2 23760.68} C_VEL
LIN {X 0,Y 505.855,Z 222.213,A -85,B 0,C 180,E1 23757.168,E2 23757.168} C_VEL
LIN {X 0,Y 505.84,Z 222.182,A -85,B 0,C 180,E1 23753.645,E2 23753.645} C_VEL
LIN {X 0,Y 505.862,Z 222.216,A -85,B 0,C 180,E1 23750.098,E2 23750.098} C_VEL
LIN {X 0,Y 505.872,Z 222.216,A -85,B 0,C 180,E1 23746.512,E2 23746.512} C_VEL
LIN {X 0,Y 505.85,Z 222.219,A -85,B 0,C 180,E1 23743.078,E2 23743.078} C_VEL
LIN {X 0,Y 505.837,Z 222.219,A -85,B 0,C 180,E1 23739.52,E2 23739.52} C_VEL
LIN {X 0,Y 505.863,Z 222.211,A -85,B 0,C 180,E1 23736.096,E2 23736.096} C_VEL
LIN {X 0,Y 505.873,Z 222.21,A -85,B 0,C 180,E1 23732.558,E2 23732.558} C_VEL
LIN {X 0,Y 505.833,Z 222.221,A -85,B 0,C 180,E1 23729.205,E2 23729.205} C_VEL
LIN {X 0,Y 505.912,Z 222.453,A -85,B 0,C 180,E1 23728.458,E2 23728.458} C_VEL
LIN {X 0,Y 507.3,Z 225.898,A -85,B 0,C 180,E1 23727.944,E2 23727.944} C_VEL
LIN {X 0,Y 508.301,Z 227.618,A -85,B 0,C 180,E1 23727.652,E2 23727.652} C_VEL
LIN {X 0,Y 513.311,Z 237.529,A -85,B 0,C 180,E1 23726.08,E2 23726.08} C_VEL
LIN {X 0,Y 521.601,Z 253.365,A -85,B 0,C 180,E1 23723.676,E2 23723.676} C_VEL
LIN {X 0,Y 532.956,Z 276.351,A -85,B 0,C 180,E1 23720.505,E2 23720.505} C_VEL
LIN {X 0,Y 544.952,Z 301.312,A -85,B 0,C 180,E1 23717.386,E2 23717.386} C_VEL
LIN {X 0,Y 547.961,Z 307.788,A -85,B 0,C 180,E1 23716.633,E2 23716.633} C_VEL
LIN {X 0,Y 547.233,Z 315.374,A -85,B 0,C 180,E1 23716.192,E2 23716.192} C_VEL
LIN {X 0,Y 550.059,Z 342.901,A -85,B 0,C 180,E1 23715.431,E2 23715.431} C_VEL
LIN {X 0,Y 541.407,Z 573.916,A -85,B 0,C 180,E1 23711.799,E2 23711.799} C_VEL
LIN {X 0,Y 537.523,Z 692.937,A -85,B 0,C 180,E1 23709.962,E2 23709.962} C_VEL
LIN {X 0,Y 535.962,Z 717.382,A -85,B 0,C 180,E1 23709.407,E2 23709.407} C_VEL
LIN {X 0,Y 534.114,Z 740.937,A -85,B 0,C 180,E1 23708.702,E2 23708.702} C_VEL
LIN {X 0,Y 531.911,Z 763.372,A -85,B 0,C 180,E1 23707.836,E2 23707.836} C_VEL
LIN {X 0,Y 529.409,Z 786.177,A -85,B 0,C 180,E1 23706.778,E2 23706.778} C_VEL
LIN {X 0,Y 526.634,Z 808.439,A -85,B 0,C 180,E1 23705.52,E2 23705.52} C_VEL
LIN {X 0,Y 523.723,Z 830.244,A -85,B 0,C 180,E1 23704.08,E2 23704.08} C_VEL
LIN {X 0,Y 521.006,Z 849.376,A -85,B 0,C 180,E1 23702.594,E2 23702.594} C_VEL
LIN {X 0,Y 518.114,Z 869.305,A -85,B 0,C 180,E1 23700.818,E2 23700.818} C_VEL
LIN {X 0,Y 515.412,Z 887.271,A -85,B 0,C 180,E1 23698.963,E2 23698.963} C_VEL
LIN {X 0,Y 512.864,Z 904.788,A -85,B 0,C 180,E1 23696.892,E2 23696.892} C_VEL
LIN {X 0,Y 510.766,Z 919.47,A -85,B 0,C 180,E1 23694.891,E2 23694.891} C_VEL
LIN {X 0,Y 508.759,Z 934.69,A -85,B 0,C 180,E1 23692.524,E2 23692.524} C_VEL
LIN {X 0,Y 507.261,Z 946.969,A -85,B 0,C 180,E1 23690.299,E2 23690.299} C_VEL
LIN {X 0,Y 506.043,Z 958.805,A -85,B 0,C 180,E1 23687.834,E2 23687.834} C_VEL
LIN {X 0,Y 505.181,Z 968.655,A -85,B 0,C 180,E1 23685.38,E2 23685.38} C_VEL
LIN {X 0,Y 504.625,Z 977.193,A -85,B 0,C 180,E1 23682.87,E2 23682.87} C_VEL
LIN {X 0,Y 504.311,Z 984.173,A -85,B 0,C 180,E1 23680.279,E2 23680.279} C_VEL
LIN {X 0,Y 504.188,Z 989.053,A -85,B 0,C 180,E1 23677.98,E2 23677.98} C_VEL
LIN {X 0,Y 504.155,Z 993.143,A -85,B 0,C 180,E1 23675.349,E2 23675.349} C_VEL
LIN {X 0,Y 504.189,Z 995.338,A -85,B 0,C 180,E1 23672.956,E2 23672.956} C_VEL
LIN {X 0,Y 504.215,Z 996.212,A -85,B 0,C 180,E1 23670.795,E2 23670.795} C_VEL
LIN {X 0,Y 504.234,Z 995.94,A -85,B 0,C 180,E1 23668.409,E2 23668.409} C_VEL
LIN {X 0,Y 504.225,Z 994.014,A -85,B 0,C 180,E1 23665.792,E2 23665.792} C_VEL
LIN {X 0,Y 504.228,Z 990.823,A -85,B 0,C 180,E1 23663.395,E2 23663.395} C_VEL
LIN {X 0,Y 504.291,Z 985.794,A -85,B 0,C 180,E1 23660.758,E2 23660.758} C_VEL
LIN {X 0,Y 504.507,Z 979.183,A -85,B 0,C 180,E1 23658.221,E2 23658.221} C_VEL
LIN {X 0,Y 504.889,Z 971.777,A -85,B 0,C 180,E1 23655.901,E2 23655.901} C_VEL
LIN {X 0,Y 505.631,Z 961.351,A -85,B 0,C 180,E1 23653.219,E2 23653.219} C_VEL
LIN {X 0,Y 506.522,Z 951.105,A -85,B 0,C 180,E1 23650.991,E2 23650.991} C_VEL
LIN {X 0,Y 507.96,Z 937.185,A -85,B 0,C 180,E1 23648.401,E2 23648.401} C_VEL
LIN {X 0,Y 509.531,Z 923.967,A -85,B 0,C 180,E1 23646.279,E2 23646.279} C_VEL
LIN {X 0,Y 511.665,Z 907.04,A -85,B 0,C 180,E1 23643.916,E2 23643.916} C_VEL
LIN {X 0,Y 513.877,Z 890.498,A -85,B 0,C 180,E1 23641.909,E2 23641.909} C_VEL
LIN {X 0,Y 516.545,Z 870.902,A -85,B 0,C 180,E1 23639.846,E2 23639.846} C_VEL
LIN {X 0,Y 519.296,Z 851.043,A -85,B 0,C 180,E1 23638.028,E2 23638.028} C_VEL
LIN {X 0,Y 522.059,Z 830.12,A -85,B 0,C 180,E1 23636.391,E2 23636.391} C_VEL
LIN {X 0,Y 524.827,Z 808.73,A -85,B 0,C 180,E1 23634.941,E2 23634.941} C_VEL
LIN {X 0,Y 527.212,Z 788.677,A -85,B 0,C 180,E1 23633.788,E2 23633.788} C_VEL
LIN {X 0,Y 529.764,Z 766.004,A -85,B 0,C 180,E1 23632.675,E2 23632.675} C_VEL
LIN {X 0,Y 531.957,Z 743.277,A -85,B 0,C 180,E1 23631.769,E2 23631.769} C_VEL
LIN {X 0,Y 533.987,Z 718.66,A -85,B 0,C 180,E1 23630.986,E2 23630.986} C_VEL
LIN {X 0,Y 535.478,Z 695.689,A -85,B 0,C 180,E1 23630.439,E2 23630.439} C_VEL
LIN {X 0,Y 536.94,Z 659.167,A -85,B 0,C 180,E1 23629.831,E2 23629.831} C_VEL
LIN {X 0,Y 540.255,Z 574.178,A -85,B 0,C 180,E1 23628.443,E2 23628.443} C_VEL
LIN {X 0,Y 544.753,Z 493.17,A -85,B 0,C 180,E1 23626.977,E2 23626.977} C_VEL
LIN {X 0,Y 550.596,Z 417.849,A -85,B 0,C 180,E1 23625.494,E2 23625.494} C_VEL
LIN {X 0,Y 557.665,Z 349.724,A -85,B 0,C 180,E1 23624.06,E2 23624.06} C_VEL
LIN {X 0,Y 559.722,Z 346.061,A -85,B 0,C 180,E1 23623.878,E2 23623.878} C_VEL
LIN {X 0,Y 568.341,Z 329.893,A -85,B 0,C 180,E1 23622.361,E2 23622.361} C_VEL
LIN {X 0,Y 569.005,Z 328.713,A -85,B 0,C 180,E1 23622.21,E2 23622.21} C_VEL
LIN {X 0,Y 569.057,Z 328.367,A -85,B 0,C 180,E1 23621.755,E2 23621.755} C_VEL
LIN {X 0,Y 568.745,Z 328.729,A -85,B 0,C 180,E1 23621.513,E2 23621.513} C_VEL
LIN {X 0,Y 558.919,Z 344.974,A -85,B 0,C 180,E1 23619.692,E2 23619.692} C_VEL
LIN {X 0,Y 550.447,Z 363.444,A -85,B 0,C 180,E1 23617.746,E2 23617.746} C_VEL
LIN {X 0,Y 543.053,Z 385.211,A -85,B 0,C 180,E1 23615.604,E2 23615.604} C_VEL
LIN {X 0,Y 542.395,Z 404.872,A -85,B 0,C 180,E1 23614.212,E2 23614.212} C_VEL
LIN {X 0,Y 542.184,Z 427.764,A -85,B 0,C 180,E1 23612.805,E2 23612.805} C_VEL
LIN {X 0,Y 542.215,Z 456.835,A -85,B 0,C 180,E1 23611.273,E2 23611.273} C_VEL
LIN {X 0,Y 542.175,Z 489.262,A -85,B 0,C 180,E1 23609.818,E2 23609.818} C_VEL
LIN {X 0,Y 541.913,Z 505.914,A -85,B 0,C 180,E1 23609.168,E2 23609.168} C_VEL
LIN {X 0,Y 530.594,Z 615.774,A -85,B 0,C 180,E1 23606.437,E2 23606.437} C_VEL
LIN {X 0,Y 524.44,Z 690.806,A -85,B 0,C 180,E1 23604.566,E2 23604.566} C_VEL
LIN {X 0,Y 522.323,Z 715.201,A -85,B 0,C 180,E1 23603.734,E2 23603.734} C_VEL
LIN {X 0,Y 520.379,Z 737.047,A -85,B 0,C 180,E1 23602.779,E2 23602.779} C_VEL
LIN {X 0,Y 518.289,Z 759.221,A -85,B 0,C 180,E1 23601.569,E2 23601.569} C_VEL
LIN {X 0,Y 516.488,Z 777.69,A -85,B 0,C 180,E1 23600.335,E2 23600.335} C_VEL
LIN {X 0,Y 514.728,Z 795.255,A -85,B 0,C 180,E1 23598.93,E2 23598.93} C_VEL
LIN {X 0,Y 513.112,Z 810.559,A -85,B 0,C 180,E1 23597.463,E2 23597.463} C_VEL
LIN {X 0,Y 511.616,Z 824.465,A -85,B 0,C 180,E1 23595.879,E2 23595.879} C_VEL
LIN {X 0,Y 510.238,Z 836.828,A -85,B 0,C 180,E1 23594.179,E2 23594.179} C_VEL
LIN {X 0,Y 509.089,Z 847.114,A -85,B 0,C 180,E1 23592.477,E2 23592.477} C_VEL
LIN {X 0,Y 508.004,Z 856.463,A -85,B 0,C 180,E1 23590.547,E2 23590.547} C_VEL
LIN {X 0,Y 507.164,Z 863.792,A -85,B 0,C 180,E1 23588.617,E2 23588.617} C_VEL
LIN {X 0,Y 506.496,Z 869.496,A -85,B 0,C 180,E1 23586.575,E2 23586.575} C_VEL
LIN {X 0,Y 506.002,Z 873.287,A -85,B 0,C 180,E1 23584.534,E2 23584.534} C_VEL
LIN {X 0,Y 505.66,Z 875.269,A -85,B 0,C 180,E1 23582.493,E2 23582.493} C_VEL
LIN {X 0,Y 505.448,Z 875.491,A -85,B 0,C 180,E1 23580.453,E2 23580.453} C_VEL
LIN {X 0,Y 505.328,Z 873.985,A -85,B 0,C 180,E1 23578.413,E2 23578.413} C_VEL
LIN {X 0,Y 505.318,Z 870.766,A -85,B 0,C 180,E1 23576.37,E2 23576.37} C_VEL
LIN {X 0,Y 505.433,Z 865.768,A -85,B 0,C 180,E1 23574.314,E2 23574.314} C_VEL
LIN {X 0,Y 505.686,Z 858.959,A -85,B 0,C 180,E1 23572.273,E2 23572.273} C_VEL
LIN {X 0,Y 506.1,Z 850.635,A -85,B 0,C 180,E1 23570.332,E2 23570.332} C_VEL
LIN {X 0,Y 506.732,Z 840.288,A -85,B 0,C 180,E1 23568.389,E2 23568.389} C_VEL
LIN {X 0,Y 507.547,Z 828.415,A -85,B 0,C 180,E1 23566.558,E2 23566.558} C_VEL
LIN {X 0,Y 508.537,Z 815.041,A -85,B 0,C 180,E1 23564.84,E2 23564.84} C_VEL
LIN {X 0,Y 509.713,Z 799.72,A -85,B 0,C 180,E1 23563.196,E2 23563.196} C_VEL
LIN {X 0,Y 511.008,Z 782.908,A -85,B 0,C 180,E1 23561.696,E2 23561.696} C_VEL
LIN {X 0,Y 512.307,Z 765.224,A -85,B 0,C 180,E1 23560.385,E2 23560.385} C_VEL
LIN {X 0,Y 513.637,Z 746.61,A -85,B 0,C 180,E1 23559.249,E2 23559.249} C_VEL
LIN {X 0,Y 514.993,Z 725.822,A -85,B 0,C 180,E1 23558.233,E2 23558.233} C_VEL
LIN {X 0,Y 516.161,Z 705.108,A -85,B 0,C 180,E1 23557.449,E2 23557.449} C_VEL
LIN {X 0,Y 517.179,Z 683.961,A -85,B 0,C 180,E1 23556.865,E2 23556.865} C_VEL
LIN {X 0,Y 523.62,Z 496.861,A -85,B 0,C 180,E1 23553.47,E2 23553.47} C_VEL
LIN {X 0,Y 518.851,Z 448.174,A -85,B 0,C 180,E1 23552.196,E2 23552.196} C_VEL
LIN {X 0,Y 522.969,Z 393.462,A -85,B 0,C 180,E1 23548.301,E2 23548.301} C_VEL
LIN {X 0,Y 526.943,Z 346.207,A -85,B 0,C 180,E1 23544.904,E2 23544.904} C_VEL
LIN {X 0,Y 531.809,Z 293.798,A -85,B 0,C 180,E1 23541.099,E2 23541.099} C_VEL
LIN {X 0,Y 532.299,Z 288.48,A -85,B 0,C 180,E1 23540.707,E2 23540.707} C_VEL
LIN {X 0,Y 524.104,Z 266.395,A -85,B 0,C 180,E1 23538.241,E2 23538.241} C_VEL
LIN {X 0,Y 518.678,Z 252.705,A -85,B 0,C 180,E1 23536.587,E2 23536.587} C_VEL
LIN {X 0,Y 520.86,Z 253.372,A -85,B 0,C 180,E1 23536.283,E2 23536.283} C_VEL
LIN {X 0,Y 522.469,Z 253.675,A -85,B 0,C 180,E1 23536.072,E2 23536.072} C_VEL
LIN {X 0,Y 530.14,Z 270.546,A -85,B 0,C 180,E1 23533.954,E2 23533.954} C_VEL
LIN {X 0,Y 537.771,Z 289.424,A -85,B 0,C 180,E1 23531.731,E2 23531.731} C_VEL
LIN {X 0,Y 542.432,Z 302.595,A -85,B 0,C 180,E1 23530.257,E2 23530.257} C_VEL
LIN {X 0,Y 541.888,Z 344.229,A -85,B 0,C 180,E1 23527.378,E2 23527.378} C_VEL
LIN {X 0,Y 541.832,Z 352.535,A -85,B 0,C 180,E1 23526.852,E2 23526.852} C_VEL
LIN {X 0,Y 539.174,Z 365.352,A -85,B 0,C 180,E1 23526.372,E2 23526.372} C_VEL
LIN {X 0,Y 538.574,Z 386.081,A -85,B 0,C 180,E1 23526.074,E2 23526.074} C_VEL
LIN {X 0,Y 537.549,Z 393.768,A -85,B 0,C 180,E1 23526.028,E2 23526.028} C_VEL
LIN {X 0,Y 531.97,Z 414.245,A -85,B 0,C 180,E1 23526.132,E2 23526.132} C_VEL
LIN {X 0,Y 531.147,Z 420.838,A -85,B 0,C 180,E1 23526.082,E2 23526.082} C_VEL
LIN {X 0,Y 528.344,Z 490.186,A -85,B 0,C 180,E1 23524.955,E2 23524.955} C_VEL
LIN {X 0,Y 524.295,Z 567.12,A -85,B 0,C 180,E1 23523.504,E2 23523.504} C_VEL
LIN {X 0,Y 520.473,Z 635.606,A -85,B 0,C 180,E1 23522.033,E2 23522.033} C_VEL
LIN {X 0,Y 519.366,Z 658.237,A -85,B 0,C 180,E1 23521.404,E2 23521.404} C_VEL
LIN {X 0,Y 517.948,Z 679.647,A -85,B 0,C 180,E1 23520.608,E2 23520.608} C_VEL
LIN {X 0,Y 516.172,Z 700.962,A -85,B 0,C 180,E1 23519.602,E2 23519.602} C_VEL
LIN {X 0,Y 514.095,Z 721.659,A -85,B 0,C 180,E1 23518.395,E2 23518.395} C_VEL
LIN {X 0,Y 511.877,Z 741.271,A -85,B 0,C 180,E1 23517.011,E2 23517.011} C_VEL
LIN {X 0,Y 509.646,Z 759.198,A -85,B 0,C 180,E1 23515.512,E2 23515.512} C_VEL
LIN {X 0,Y 507.324,Z 776.844,A -85,B 0,C 180,E1 23513.769,E2 23513.769} C_VEL
LIN {X 0,Y 505.075,Z 793.275,A -85,B 0,C 180,E1 23511.85,E2 23511.85} C_VEL
LIN {X 0,Y 502.998,Z 808.447,A -85,B 0,C 180,E1 23509.751,E2 23509.751} C_VEL
LIN {X 0,Y 501.291,Z 821.269,A -85,B 0,C 180,E1 23507.649,E2 23507.649} C_VEL
LIN {X 0,Y 499.859,Z 832.688,A -85,B 0,C 180,E1 23505.429,E2 23505.429} C_VEL
LIN {X 0,Y 498.729,Z 842.666,A -85,B 0,C 180,E1 23503.094,E2 23503.094} C_VEL
LIN {X 0,Y 497.931,Z 850.784,A -85,B 0,C 180,E1 23500.763,E2 23500.763} C_VEL
LIN {X 0,Y 497.386,Z 857.452,A -85,B 0,C 180,E1 23498.322,E2 23498.322} C_VEL
LIN {X 0,Y 497.063,Z 862.275,A -85,B 0,C 180,E1 23495.889,E2 23495.889} C_VEL
LIN {X 0,Y 496.894,Z 865.442,A -85,B 0,C 180,E1 23493.461,E2 23493.461} C_VEL
LIN {X 0,Y 496.823,Z 867.011,A -85,B 0,C 180,E1 23491.038,E2 23491.038} C_VEL
LIN {X 0,Y 496.828,Z 866.984,A -85,B 0,C 180,E1 23488.732,E2 23488.732} C_VEL
LIN {X 0,Y 496.892,Z 865.419,A -85,B 0,C 180,E1 23486.424,E2 23486.424} C_VEL
LIN {X 0,Y 497.066,Z 862.234,A -85,B 0,C 180,E1 23483.996,E2 23483.996} C_VEL
LIN {X 0,Y 497.391,Z 857.399,A -85,B 0,C 180,E1 23481.561,E2 23481.561} C_VEL
LIN {X 0,Y 497.95,Z 850.629,A -85,B 0,C 180,E1 23479.09,E2 23479.09} C_VEL
LIN {X 0,Y 498.743,Z 842.577,A -85,B 0,C 180,E1 23476.788,E2 23476.788} C_VEL
LIN {X 0,Y 499.878,Z 832.577,A -85,B 0,C 180,E1 23474.453,E2 23474.453} C_VEL
LIN {X 0,Y 501.315,Z 821.132,A -85,B 0,C 180,E1 23472.232,E2 23472.232} C_VEL
LIN {X 0,Y 503.031,Z 808.281,A -85,B 0,C 180,E1 23470.129,E2 23470.129} C_VEL
LIN {X 0,Y 504.99,Z 793.993,A -85,B 0,C 180,E1 23468.146,E2 23468.146} C_VEL
LIN {X 0,Y 507.146,Z 778.179,A -85,B 0,C 180,E1 23466.284,E2 23466.284} C_VEL
LIN {X 0,Y 509.359,Z 761.425,A -85,B 0,C 180,E1 23464.601,E2 23464.601} C_VEL
LIN {X 0,Y 511.671,Z 743.145,A -85,B 0,C 180,E1 23463.04,E2 23463.04} C_VEL
LIN {X 0,Y 513.878,Z 723.908,A -85,B 0,C 180,E1 23461.656,E2 23461.656} C_VEL
LIN {X 0,Y 515.863,Z 704.567,A -85,B 0,C 180,E1 23460.493,E2 23460.493} C_VEL
LIN {X 0,Y 517.689,Z 683.844,A -85,B 0,C 180,E1 23459.471,E2 23459.471} C_VEL
LIN {X 0,Y 519.229,Z 661.611,A -85,B 0,C 180,E1 23458.607,E2 23458.607} C_VEL
LIN {X 0,Y 520.365,Z 638.867,A -85,B 0,C 180,E1 23457.95,E2 23457.95} C_VEL
LIN {X 0,Y 523.744,Z 577.359,A -85,B 0,C 180,E1 23456.608,E2 23456.608} C_VEL
LIN {X 0,Y 527.915,Z 499.903,A -85,B 0,C 180,E1 23455.123,E2 23455.123} C_VEL
LIN {X 0,Y 530.827,Z 431.423,A -85,B 0,C 180,E1 23453.983,E2 23453.983} C_VEL
LIN {X 0,Y 532.847,Z 366.95,A -85,B 0,C 180,E1 23453.028,E2 23453.028} C_VEL
LIN {X 0,Y 535.831,Z 353.175,A -85,B 0,C 180,E1 23452.474,E2 23452.474} C_VEL
LIN {X 0,Y 536.059,Z 315.952,A -85,B 0,C 180,E1 23449.946,E2 23449.946} C_VEL
LIN {X 0,Y 536.161,Z 305.817,A -85,B 0,C 180,E1 23449.214,E2 23449.214} C_VEL
LIN {X 0,Y 528.346,Z 284.769,A -85,B 0,C 180,E1 23446.77,E2 23446.77} C_VEL
LIN {X 0,Y 520.091,Z 265.604,A -85,B 0,C 180,E1 23444.411,E2 23444.411} C_VEL
LIN {X 0,Y 511.867,Z 248.983,A -85,B 0,C 180,E1 23442.22,E2 23442.22} C_VEL
LIN {X 0,Y 505.146,Z 236.611,A -85,B 0,C 180,E1 23440.485,E2 23440.485} C_VEL
LIN {X 0,Y 502.582,Z 232.134,A -85,B 0,C 180,E1 23439.838,E2 23439.838} C_VEL
LIN {X 0,Y 500.537,Z 228.181,A -85,B 0,C 180,E1 23439.291,E2 23439.291} C_VEL
LIN {X 0,Y 498.69,Z 225.789,A -85,B 0,C 180,E1 23438.872,E2 23438.872} C_VEL
LIN {X 0,Y 497.917,Z 223.213,A -85,B 0,C 180,E1 23438.559,E2 23438.559} C_VEL
LIN {X 0,Y 497.916,Z 223.21,A -85,B 0,C 180,E1 23434.913,E2 23434.913} C_VEL
LIN {X 0,Y 497.931,Z 223.201,A -85,B 0,C 180,E1 23431.339,E2 23431.339} C_VEL
LIN {X 0,Y 497.921,Z 223.181,A -85,B 0,C 180,E1 23427.768,E2 23427.768} C_VEL
LIN {X 0,Y 497.924,Z 223.174,A -85,B 0,C 180,E1 23424.183,E2 23424.183} C_VEL
LIN {X 0,Y 497.923,Z 223.206,A -85,B 0,C 180,E1 23420.645,E2 23420.645} C_VEL
LIN {X 0,Y 497.924,Z 223.176,A -85,B 0,C 180,E1 23417.049,E2 23417.049} C_VEL
LIN {X 0,Y 497.914,Z 223.184,A -85,B 0,C 180,E1 23413.589,E2 23413.589} C_VEL
LIN {X 0,Y 497.919,Z 223.2,A -85,B 0,C 180,E1 23409.945,E2 23409.945} C_VEL
LIN {X 0,Y 497.924,Z 223.166,A -85,B 0,C 180,E1 23406.457,E2 23406.457} C_VEL
LIN {X 0,Y 497.926,Z 223.205,A -85,B 0,C 180,E1 23402.878,E2 23402.878} C_VEL
LIN {X 0,Y 497.905,Z 223.163,A -85,B 0,C 180,E1 23399.425,E2 23399.425} C_VEL
LIN {X 0,Y 497.911,Z 223.208,A -85,B 0,C 180,E1 23395.854,E2 23395.854} C_VEL
LIN {X 0,Y 497.927,Z 223.163,A -85,B 0,C 180,E1 23392.268,E2 23392.268} C_VEL
LIN {X 0,Y 497.93,Z 223.205,A -85,B 0,C 180,E1 23388.65,E2 23388.65} C_VEL
LIN {X 0,Y 497.908,Z 223.202,A -85,B 0,C 180,E1 23385.105,E2 23385.105} C_VEL
LIN {X 0,Y 497.901,Z 223.2,A -85,B 0,C 180,E1 23381.622,E2 23381.622} C_VEL
LIN {X 0,Y 497.926,Z 223.2,A -85,B 0,C 180,E1 23378.068,E2 23378.068} C_VEL
LIN {X 0,Y 497.932,Z 223.207,A -85,B 0,C 180,E1 23374.549,E2 23374.549} C_VEL
LIN {X 0,Y 497.904,Z 223.202,A -85,B 0,C 180,E1 23371.054,E2 23371.054} C_VEL
LIN {X 0,Y 497.895,Z 223.235,A -85,B 0,C 180,E1 23369.464,E2 23369.464} C_VEL
LIN {X 0,Y 498.983,Z 226.339,A -85,B 0,C 180,E1 23369.003,E2 23369.003} C_VEL
LIN {X 0,Y 500.209,Z 227.869,A -85,B 0,C 180,E1 23368.686,E2 23368.686} C_VEL
LIN {X 0,Y 502.184,Z 232.043,A -85,B 0,C 180,E1 23368.017,E2 23368.017} C_VEL
LIN {X 0,Y 511.698,Z 250.645,A -85,B 0,C 180,E1 23365.072,E2 23365.072} C_VEL
LIN {X 0,Y 521.909,Z 270.924,A -85,B 0,C 180,E1 23362.122,E2 23362.122} C_VEL
LIN {X 0,Y 533.419,Z 294.639,A -85,B 0,C 180,E1 23358.999,E2 23358.999} C_VEL
LIN {X 0,Y 541.259,Z 311.648,A -85,B 0,C 180,E1 23356.963,E2 23356.963} C_VEL
LIN {X 0,Y 540.884,Z 316.257,A -85,B 0,C 180,E1 23356.708,E2 23356.708} C_VEL
LIN {X 0,Y 543.669,Z 344.055,A -85,B 0,C 180,E1 23355.925,E2 23355.925} C_VEL
LIN {X 0,Y 534.333,Z 582.812,A -85,B 0,C 180,E1 23352.117,E2 23352.117} C_VEL
LIN {X 0,Y 530.588,Z 692.929,A -85,B 0,C 180,E1 23350.391,E2 23350.391} C_VEL
LIN {X 0,Y 528.963,Z 717.488,A -85,B 0,C 180,E1 23349.826,E2 23349.826} C_VEL
LIN {X 0,Y 527.05,Z 741.067,A -85,B 0,C 180,E1 23349.11,E2 23349.11} C_VEL
LIN {X 0,Y 524.741,Z 763.853,A -85,B 0,C 180,E1 23348.217,E2 23348.217} C_VEL
LIN {X 0,Y 522.207,Z 786.241,A -85,B 0,C 180,E1 23347.164,E2 23347.164} C_VEL
LIN {X 0,Y 519.472,Z 807.492,A -85,B 0,C 180,E1 23345.949,E2 23345.949} C_VEL
LIN {X 0,Y 516.575,Z 828.598,A -85,B 0,C 180,E1 23344.551,E2 23344.551} C_VEL
LIN {X 0,Y 513.566,Z 849.024,A -85,B 0,C 180,E1 23342.95,E2 23342.95} C_VEL
LIN {X 0,Y 510.552,Z 869.166,A -85,B 0,C 180,E1 23341.133,E2 23341.133} C_VEL
LIN {X 0,Y 507.908,Z 886.18,A -85,B 0,C 180,E1 23339.353,E2 23339.353} C_VEL
LIN {X 0,Y 505.186,Z 904.141,A -85,B 0,C 180,E1 23337.207,E2 23337.207} C_VEL
LIN {X 0,Y 503.016,Z 918.875,A -85,B 0,C 180,E1 23335.175,E2 23335.175} C_VEL
LIN {X 0,Y 501.019,Z 933.36,A -85,B 0,C 180,E1 23332.902,E2 23332.902} C_VEL
LIN {X 0,Y 499.372,Z 946.381,A -85,B 0,C 180,E1 23330.512,E2 23330.512} C_VEL
LIN {X 0,Y 498.108,Z 958.222,A -85,B 0,C 180,E1 23328.007,E2 23328.007} C_VEL
LIN {X 0,Y 497.216,Z 968.061,A -85,B 0,C 180,E1 23325.513,E2 23325.513} C_VEL
LIN {X 0,Y 496.64,Z 976.729,A -85,B 0,C 180,E1 23322.913,E2 23322.913} C_VEL
LIN {X 0,Y 496.324,Z 983.79,A -85,B 0,C 180,E1 23320.212,E2 23320.212} C_VEL
LIN {X 0,Y 496.196,Z 988.809,A -85,B 0,C 180,E1 23317.759,E2 23317.759} C_VEL
LIN {X 0,Y 496.201,Z 992.633,A -85,B 0,C 180,E1 23315.087,E2 23315.087} C_VEL
LIN {X 0,Y 496.232,Z 994.538,A -85,B 0,C 180,E1 23312.887,E2 23312.887} C_VEL
LIN {X 0,Y 496.261,Z 995.356,A -85,B 0,C 180,E1 23310.693,E2 23310.693} C_VEL
LIN {X 0,Y 496.28,Z 994.989,A -85,B 0,C 180,E1 23308.153,E2 23308.153} C_VEL
LIN {X 0,Y 496.266,Z 992.974,A -85,B 0,C 180,E1 23305.609,E2 23305.609} C_VEL
LIN {X 0,Y 496.267,Z 989.888,A -85,B 0,C 180,E1 23303.289,E2 23303.289} C_VEL
LIN {X 0,Y 496.332,Z 984.812,A -85,B 0,C 180,E1 23300.608,E2 23300.608} C_VEL
LIN {X 0,Y 496.549,Z 978.157,A -85,B 0,C 180,E1 23298.029,E2 23298.029} C_VEL
LIN {X 0,Y 496.949,Z 970.715,A -85,B 0,C 180,E1 23295.671,E2 23295.671} C_VEL
LIN {X 0,Y 497.723,Z 960.221,A -85,B 0,C 180,E1 23292.944,E2 23292.944} C_VEL
LIN {X 0,Y 498.668,Z 949.927,A -85,B 0,C 180,E1 23290.68,E2 23290.68} C_VEL
LIN {X 0,Y 500.185,Z 935.955,A -85,B 0,C 180,E1 23288.048,E2 23288.048} C_VEL
LIN {X 0,Y 501.854,Z 922.46,A -85,B 0,C 180,E1 23285.856,E2 23285.856} C_VEL
LIN {X 0,Y 504.143,Z 905.307,A -85,B 0,C 180,E1 23283.444,E2 23283.444} C_VEL
LIN {X 0,Y 506.492,Z 888.608,A -85,B 0,C 180,E1 23281.397,E2 23281.397} C_VEL
LIN {X 0,Y 509.252,Z 869.46,A -85,B 0,C 180,E1 23279.368,E2 23279.368} C_VEL
LIN {X 0,Y 512.045,Z 850.249,A -85,B 0,C 180,E1 23277.586,E2 23277.586} C_VEL
LIN {X 0,Y 514.947,Z 829.398,A -85,B 0,C 180,E1 23275.931,E2 23275.931} C_VEL
LIN {X 0,Y 517.868,Z 808.115,A -85,B 0,C 180,E1 23274.467,E2 23274.467} C_VEL
LIN {X 0,Y 520.458,Z 787.463,A -85,B 0,C 180,E1 23273.264,E2 23273.264} C_VEL
LIN {X 0,Y 523.114,Z 765.032,A -85,B 0,C 180,E1 23272.152,E2 23272.152} C_VEL
LIN {X 0,Y 525.438,Z 742.393,A -85,B 0,C 180,E1 23271.239,E2 23271.239} C_VEL
LIN {X 0,Y 527.646,Z 716.844,A -85,B 0,C 180,E1 23270.42,E2 23270.42} C_VEL
LIN {X 0,Y 529.391,Z 692.114,A -85,B 0,C 180,E1 23269.833,E2 23269.833} C_VEL
LIN {X 0,Y 534.165,Z 581.206,A -85,B 0,C 180,E1 23267.968,E2 23267.968} C_VEL
LIN {X 0,Y 538.929,Z 503.389,A -85,B 0,C 180,E1 23266.52,E2 23266.52} C_VEL
LIN {X 0,Y 545.076,Z 430.601,A -85,B 0,C 180,E1 23265.046,E2 23265.046} C_VEL
LIN {X 0,Y 552.742,Z 362.529,A -85,B 0,C 180,E1 23263.581,E2 23263.581} C_VEL
LIN {X 0,Y 554.177,Z 352.559,A -85,B 0,C 180,E1 23263.354,E2 23263.354} C_VEL
LIN {X 0,Y 556.507,Z 348.629,A -85,B 0,C 180,E1 23263.158,E2 23263.158} C_VEL
LIN {X 0,Y 564.301,Z 335.308,A -85,B 0,C 180,E1 23261.868,E2 23261.868} C_VEL
LIN {X 0,Y 554.245,Z 350.827,A -85,B 0,C 180,E1 23260.095,E2 23260.095} C_VEL
LIN {X 0,Y 545.277,Z 369.18,A -85,B 0,C 180,E1 23258.124,E2 23258.124} C_VEL
LIN {X 0,Y 541.272,Z 380.071,A -85,B 0,C 180,E1 23257.029,E2 23257.029} C_VEL
LIN {X 0,Y 539.882,Z 395.489,A -85,B 0,C 180,E1 23255.811,E2 23255.811} C_VEL
LIN {X 0,Y 538.901,Z 414.359,A -85,B 0,C 180,E1 23254.492,E2 23254.492} C_VEL
LIN {X 0,Y 538.23,Z 436.085,A -85,B 0,C 180,E1 23253.177,E2 23253.177} C_VEL
LIN {X 0,Y 537.746,Z 462.687,A -85,B 0,C 180,E1 23251.767,E2 23251.767} C_VEL
LIN {X 0,Y 537.226,Z 494.399,A -85,B 0,C 180,E1 23250.322,E2 23250.322} C_VEL
LIN {X 0,Y 536.808,Z 507.507,A -85,B 0,C 180,E1 23249.804,E2 23249.804} C_VEL
LIN {X 0,Y 525.195,Z 612.307,A -85,B 0,C 180,E1 23247.135,E2 23247.135} C_VEL
LIN {X 0,Y 518.134,Z 690.947,A -85,B 0,C 180,E1 23245.111,E2 23245.111} C_VEL
LIN {X 0,Y 515.856,Z 715.335,A -85,B 0,C 180,E1 23244.263,E2 23244.263} C_VEL
LIN {X 0,Y 513.695,Z 737.418,A -85,B 0,C 180,E1 23243.274,E2 23243.274} C_VEL
LIN {X 0,Y 511.583,Z 758.559,A -85,B 0,C 180,E1 23242.114,E2 23242.114} C_VEL
LIN {X 0,Y 509.453,Z 778.751,A -85,B 0,C 180,E1 23240.748,E2 23240.748} C_VEL
LIN {X 0,Y 507.637,Z 795.554,A -85,B 0,C 180,E1 23239.384,E2 23239.384} C_VEL
LIN {X 0,Y 505.847,Z 811.517,A -85,B 0,C 180,E1 23237.841,E2 23237.841} C_VEL
LIN {X 0,Y 504.229,Z 825.364,A -85,B 0,C 180,E1 23236.237,E2 23236.237} C_VEL
LIN {X 0,Y 502.759,Z 837.804,A -85,B 0,C 180,E1 23234.512,E2 23234.512} C_VEL
LIN {X 0,Y 501.427,Z 848.665,A -85,B 0,C 180,E1 23232.671,E2 23232.671} C_VEL
LIN {X 0,Y 500.343,Z 857.501,A -85,B 0,C 180,E1 23230.827,E2 23230.827} C_VEL
LIN {X 0,Y 499.418,Z 864.812,A -85,B 0,C 180,E1 23228.868,E2 23228.868} C_VEL
LIN {X 0,Y 498.69,Z 870.567,A -85,B 0,C 180,E1 23226.794,E2 23226.794} C_VEL
LIN {X 0,Y 498.146,Z 874.376,A -85,B 0,C 180,E1 23224.721,E2 23224.721} C_VEL
LIN {X 0,Y 497.766,Z 876.362,A -85,B 0,C 180,E1 23222.648,E2 23222.648} C_VEL
LIN {X 0,Y 497.53,Z 876.601,A -85,B 0,C 180,E1 23220.576,E2 23220.576} C_VEL
LIN {X 0,Y 497.397,Z 875.104,A -85,B 0,C 180,E1 23218.502,E2 23218.502} C_VEL
LIN {X 0,Y 497.377,Z 871.889,A -85,B 0,C 180,E1 23216.427,E2 23216.427} C_VEL
LIN {X 0,Y 497.487,Z 866.903,A -85,B 0,C 180,E1 23214.348,E2 23214.348} C_VEL
LIN {X 0,Y 497.726,Z 860.486,A -85,B 0,C 180,E1 23212.381,E2 23212.381} C_VEL
LIN {X 0,Y 498.141,Z 852.263,A -85,B 0,C 180,E1 23210.41,E2 23210.41} C_VEL
LIN {X 0,Y 498.775,Z 842.028,A -85,B 0,C 180,E1 23208.436,E2 23208.436} C_VEL
LIN {X 0,Y 499.598,Z 830.284,A -85,B 0,C 180,E1 23206.576,E2 23206.576} C_VEL
LIN {X 0,Y 500.6,Z 817.064,A -85,B 0,C 180,E1 23204.831,E2 23204.831} C_VEL
LIN {X 0,Y 501.788,Z 802.012,A -85,B 0,C 180,E1 23203.168,E2 23203.168} C_VEL
LIN {X 0,Y 503.112,Z 785.453,A -85,B 0,C 180,E1 23201.639,E2 23201.639} C_VEL
LIN {X 0,Y 504.503,Z 767.326,A -85,B 0,C 180,E1 23200.25,E2 23200.25} C_VEL
LIN {X 0,Y 505.928,Z 747.989,A -85,B 0,C 180,E1 23199.04,E2 23199.04} C_VEL
LIN {X 0,Y 507.242,Z 728.723,A -85,B 0,C 180,E1 23198.065,E2 23198.065} C_VEL
LIN {X 0,Y 508.498,Z 707.478,A -85,B 0,C 180,E1 23197.226,E2 23197.226} C_VEL
LIN {X 0,Y 509.582,Z 686,A -85,B 0,C 180,E1 23196.603,E2 23196.603} C_VEL
LIN {X 0,Y 510.841,Z 649.884,A -85,B 0,C 180,E1 23195.903,E2 23195.903} C_VEL
LIN {X 0,Y 516.396,Z 497.59,A -85,B 0,C 180,E1 23193.092,E2 23193.092} C_VEL
LIN {X 0,Y 511.577,Z 447.124,A -85,B 0,C 180,E1 23191.739,E2 23191.739} C_VEL
LIN {X 0,Y 515.756,Z 394.023,A -85,B 0,C 180,E1 23187.909,E2 23187.909} C_VEL
LIN {X 0,Y 519.879,Z 347.002,A -85,B 0,C 180,E1 23184.49,E2 23184.49} C_VEL
LIN {X 0,Y 524.881,Z 295.349,A -85,B 0,C 180,E1 23180.698,E2 23180.698} C_VEL
LIN {X 0,Y 525.082,Z 291.057,A -85,B 0,C 180,E1 23180.362,E2 23180.362} C_VEL
LIN {X 0,Y 516.748,Z 268.716,A -85,B 0,C 180,E1 23177.822,E2 23177.822} C_VEL
LIN {X 0,Y 513.337,Z 259.733,A -85,B 0,C 180,E1 23176.714,E2 23176.714} C_VEL
LIN {X 0,Y 515.183,Z 260.362,A -85,B 0,C 180,E1 23176.449,E2 23176.449} C_VEL
LIN {X 0,Y 517.808,Z 260.741,A -85,B 0,C 180,E1 23176.113,E2 23176.113} C_VEL
LIN {X 0,Y 525.294,Z 277.616,A -85,B 0,C 180,E1 23173.985,E2 23173.985} C_VEL
LIN {X 0,Y 532.91,Z 297.004,A -85,B 0,C 180,E1 23171.689,E2 23171.689} C_VEL
LIN {X 0,Y 536.205,Z 306.454,A -85,B 0,C 180,E1 23170.627,E2 23170.627} C_VEL
LIN {X 0,Y 535.707,Z 348.21,A -85,B 0,C 180,E1 23167.749,E2 23167.749} C_VEL
LIN {X 0,Y 535.539,Z 354.533,A -85,B 0,C 180,E1 23167.359,E2 23167.359} C_VEL
LIN {X 0,Y 532.735,Z 368.037,A -85,B 0,C 180,E1 23166.855,E2 23166.855} C_VEL
LIN {X 0,Y 531.147,Z 420.838,A -85,B 0,C 180,E1 23166.082,E2 23166.082} C_VEL
LIN {X 0,Y 530.074,Z 428.519,A -85,B 0,C 180,E1 23166.032,E2 23166.032} C_VEL
LIN {X 0,Y 524.319,Z 448.958,A -85,B 0,C 180,E1 23166.126,E2 23166.126} C_VEL
LIN {X 0,Y 523.463,Z 455.536,A -85,B 0,C 180,E1 23166.066,E2 23166.066} C_VEL
LIN {X 0,Y 519.987,Z 527.674,A -85,B 0,C 180,E1 23164.786,E2 23164.786} C_VEL
LIN {X 0,Y 515.254,Z 607.323,A -85,B 0,C 180,E1 23163.157,E2 23163.157} C_VEL
LIN {X 0,Y 513.124,Z 648.267,A -85,B 0,C 180,E1 23162.185,E2 23162.185} C_VEL
LIN {X 0,Y 511.85,Z 670.06,A -85,B 0,C 180,E1 23161.471,E2 23161.471} C_VEL
LIN {X 0,Y 510.196,Z 691.298,A -85,B 0,C 180,E1 23160.569,E2 23160.569} C_VEL
LIN {X 0,Y 508.197,Z 712.118,A -85,B 0,C 180,E1 23159.464,E2 23159.464} C_VEL
LIN {X 0,Y 506.025,Z 731.949,A -85,B 0,C 180,E1 23158.181,E2 23158.181} C_VEL
LIN {X 0,Y 503.772,Z 750.161,A -85,B 0,C 180,E1 23156.779,E2 23156.779} C_VEL
LIN {X 0,Y 501.33,Z 768.422,A -85,B 0,C 180,E1 23155.11,E2 23155.11} C_VEL
LIN {X 0,Y 498.97,Z 785.034,A -85,B 0,C 180,E1 23153.314,E2 23153.314} C_VEL
LIN {X 0,Y 496.886,Z 799.497,A -85,B 0,C 180,E1 23151.484,E2 23151.484} C_VEL
LIN {X 0,Y 494.823,Z 813.874,A -85,B 0,C 180,E1 23149.354,E2 23149.354} C_VEL
LIN {X 0,Y 493.063,Z 826.677,A -85,B 0,C 180,E1 23147.101,E2 23147.101} C_VEL
LIN {X 0,Y 491.688,Z 837.411,A -85,B 0,C 180,E1 23144.847,E2 23144.847} C_VEL
LIN {X 0,Y 490.619,Z 846.749,A -85,B 0,C 180,E1 23142.476,E2 23142.476} C_VEL
LIN {X 0,Y 489.836,Z 854.52,A -85,B 0,C 180,E1 23139.992,E2 23139.992} C_VEL
LIN {X 0,Y 489.348,Z 860.2,A -85,B 0,C 180,E1 23137.632,E2 23137.632} C_VEL
LIN {X 0,Y 489.076,Z 864.511,A -85,B 0,C 180,E1 23135.161,E2 23135.161} C_VEL
LIN {X 0,Y 488.935,Z 867.192,A -85,B 0,C 180,E1 23132.696,E2 23132.696} C_VEL
LIN {X 0,Y 488.889,Z 868.168,A -85,B 0,C 180,E1 23130.234,E2 23130.234} C_VEL
LIN {X 0,Y 488.916,Z 867.511,A -85,B 0,C 180,E1 23127.773,E2 23127.773} C_VEL
LIN {X 0,Y 489.04,Z 865.259,A -85,B 0,C 180,E1 23125.309,E2 23125.309} C_VEL
LIN {X 0,Y 489.284,Z 861.392,A -85,B 0,C 180,E1 23122.839,E2 23122.839} C_VEL
LIN {X 0,Y 489.72,Z 855.73,A -85,B 0,C 180,E1 23120.362,E2 23120.362} C_VEL
LIN {X 0,Y 490.421,Z 848.634,A -85,B 0,C 180,E1 23117.997,E2 23117.997} C_VEL
LIN {X 0,Y 491.458,Z 839.295,A -85,B 0,C 180,E1 23115.508,E2 23115.508} C_VEL
LIN {X 0,Y 492.775,Z 828.984,A -85,B 0,C 180,E1 23113.254,E2 23113.254} C_VEL
LIN {X 0,Y 494.367,Z 817.386,A -85,B 0,C 180,E1 23111.119,E2 23111.119} C_VEL
LIN {X 0,Y 496.446,Z 802.797,A -85,B 0,C 180,E1 23108.868,E2 23108.868} C_VEL
LIN {X 0,Y 498.742,Z 786.853,A -85,B 0,C 180,E1 23106.8,E2 23106.8} C_VEL
LIN {X 0,Y 501.156,Z 769.789,A -85,B 0,C 180,E1 23104.933,E2 23104.933} C_VEL
LIN {X 0,Y 503.469,Z 752.531,A -85,B 0,C 180,E1 23103.331,E2 23103.331} C_VEL
LIN {X 0,Y 505.808,Z 733.895,A -85,B 0,C 180,E1 23101.864,E2 23101.864} C_VEL
LIN {X 0,Y 508.074,Z 713.598,A -85,B 0,C 180,E1 23100.528,E2 23100.528} C_VEL
LIN {X 0,Y 510.065,Z 693.123,A -85,B 0,C 180,E1 23099.423,E2 23099.423} C_VEL
LIN {X 0,Y 511.731,Z 672.225,A -85,B 0,C 180,E1 23098.513,E2 23098.513} C_VEL
LIN {X 0,Y 513.065,Z 650.65,A -85,B 0,C 180,E1 23097.784,E2 23097.784} C_VEL
LIN {X 0,Y 515.022,Z 611.532,A -85,B 0,C 180,E1 23096.838,E2 23096.838} C_VEL
LIN {X 0,Y 519.861,Z 530.594,A -85,B 0,C 180,E1 23095.175,E2 23095.175} C_VEL
LIN {X 0,Y 523.366,Z 458.843,A -85,B 0,C 180,E1 23093.893,E2 23093.893} C_VEL
LIN {X 0,Y 526.252,Z 374.974,A -85,B 0,C 180,E1 23092.616,E2 23092.616} C_VEL
LIN {X 0,Y 526.568,Z 369.122,A -85,B 0,C 180,E1 23092.512,E2 23092.512} C_VEL
LIN {X 0,Y 529.673,Z 354.611,A -85,B 0,C 180,E1 23091.924,E2 23091.924} C_VEL
LIN {X 0,Y 529.967,Z 316.559,A -85,B 0,C 180,E1 23089.329,E2 23089.329} C_VEL
LIN {X 0,Y 529.934,Z 309.573,A -85,B 0,C 180,E1 23088.814,E2 23088.814} C_VEL
LIN {X 0,Y 522.461,Z 289.382,A -85,B 0,C 180,E1 23086.451,E2 23086.451} C_VEL
LIN {X 0,Y 513.927,Z 269.463,A -85,B 0,C 180,E1 23083.956,E2 23083.956} C_VEL
LIN {X 0,Y 505.067,Z 251.535,A -85,B 0,C 180,E1 23081.545,E2 23081.545} C_VEL
LIN {X 0,Y 497.989,Z 238.548,A -85,B 0,C 180,E1 23079.68,E2 23079.68} C_VEL
LIN {X 0,Y 495.018,Z 233.573,A -85,B 0,C 180,E1 23078.917,E2 23078.917} C_VEL
LIN {X 0,Y 492.968,Z 229.775,A -85,B 0,C 180,E1 23078.365,E2 23078.365} C_VEL
LIN {X 0,Y 490.723,Z 226.675,A -85,B 0,C 180,E1 23077.83,E2 23077.83} C_VEL
LIN {X 0,Y 489.99,Z 224.177,A -85,B 0,C 180,E1 23077.519,E2 23077.519} C_VEL
LIN {X 0,Y 489.986,Z 224.18,A -85,B 0,C 180,E1 23073.996,E2 23073.996} C_VEL
LIN {X 0,Y 489.995,Z 224.192,A -85,B 0,C 180,E1 23070.325,E2 23070.325} C_VEL
LIN {X 0,Y 489.98,Z 224.188,A -85,B 0,C 180,E1 23066.807,E2 23066.807} C_VEL
LIN {X 0,Y 489.987,Z 224.157,A -85,B 0,C 180,E1 23063.194,E2 23063.194} C_VEL
LIN {X 0,Y 489.981,Z 224.179,A -85,B 0,C 180,E1 23059.677,E2 23059.677} C_VEL
LIN {X 0,Y 489.985,Z 224.184,A -85,B 0,C 180,E1 23056.023,E2 23056.023} C_VEL
LIN {X 0,Y 489.981,Z 224.153,A -85,B 0,C 180,E1 23052.493,E2 23052.493} C_VEL
LIN {X 0,Y 489.989,Z 224.194,A -85,B 0,C 180,E1 23048.922,E2 23048.922} C_VEL
LIN {X 0,Y 489.972,Z 224.156,A -85,B 0,C 180,E1 23045.386,E2 23045.386} C_VEL
LIN {X 0,Y 489.972,Z 224.189,A -85,B 0,C 180,E1 23041.754,E2 23041.754} C_VEL
LIN {X 0,Y 489.984,Z 224.161,A -85,B 0,C 180,E1 23038.246,E2 23038.246} C_VEL
LIN {X 0,Y 489.988,Z 224.178,A -85,B 0,C 180,E1 23034.731,E2 23034.731} C_VEL
LIN {X 0,Y 489.967,Z 224.171,A -85,B 0,C 180,E1 23031.314,E2 23031.314} C_VEL
LIN {X 0,Y 489.968,Z 224.198,A -85,B 0,C 180,E1 23027.747,E2 23027.747} C_VEL
LIN {X 0,Y 489.992,Z 224.186,A -85,B 0,C 180,E1 23024.252,E2 23024.252} C_VEL
LIN {X 0,Y 489.992,Z 224.189,A -85,B 0,C 180,E1 23020.696,E2 23020.696} C_VEL
LIN {X 0,Y 489.963,Z 224.2,A -85,B 0,C 180,E1 23017.186,E2 23017.186} C_VEL
LIN {X 0,Y 489.96,Z 224.191,A -85,B 0,C 180,E1 23013.584,E2 23013.584} C_VEL
LIN {X 0,Y 490.002,Z 224.209,A -85,B 0,C 180,E1 23010.462,E2 23010.462} C_VEL
LIN {X 0,Y 491.217,Z 227.578,A -85,B 0,C 180,E1 23009.951,E2 23009.951} C_VEL
LIN {X 0,Y 492.371,Z 229.242,A -85,B 0,C 180,E1 23009.625,E2 23009.625} C_VEL
LIN {X 0,Y 494.359,Z 233.153,A -85,B 0,C 180,E1 23008.951,E2 23008.951} C_VEL
LIN {X 0,Y 504.126,Z 252.236,A -85,B 0,C 180,E1 23005.854,E2 23005.854} C_VEL
LIN {X 0,Y 514.417,Z 272.721,A -85,B 0,C 180,E1 23002.807,E2 23002.807} C_VEL
LIN {X 0,Y 525.439,Z 295.438,A -85,B 0,C 180,E1 22999.737,E2 22999.737} C_VEL
LIN {X 0,Y 534.591,Z 314.923,A -85,B 0,C 180,E1 22997.333,E2 22997.333} C_VEL
LIN {X 0,Y 534.669,Z 318.06,A -85,B 0,C 180,E1 22997.209,E2 22997.209} C_VEL
LIN {X 0,Y 537.329,Z 345.264,A -85,B 0,C 180,E1 22996.432,E2 22996.432} C_VEL
LIN {X 0,Y 527.676,Z 580.872,A -85,B 0,C 180,E1 22992.617,E2 22992.617} C_VEL
LIN {X 0,Y 523.674,Z 692.969,A -85,B 0,C 180,E1 22990.83,E2 22990.83} C_VEL
LIN {X 0,Y 521.999,Z 717.336,A -85,B 0,C 180,E1 22990.26,E2 22990.26} C_VEL
LIN {X 0,Y 520.001,Z 741.084,A -85,B 0,C 180,E1 22989.529,E2 22989.529} C_VEL
LIN {X 0,Y 517.579,Z 764.203,A -85,B 0,C 180,E1 22988.608,E2 22988.608} C_VEL
LIN {X 0,Y 514.823,Z 787.471,A -85,B 0,C 180,E1 22987.485,E2 22987.485} C_VEL
LIN {X 0,Y 512.067,Z 808.281,A -85,B 0,C 180,E1 22986.274,E2 22986.274} C_VEL
LIN {X 0,Y 508.957,Z 830.059,A -85,B 0,C 180,E1 22984.795,E2 22984.795} C_VEL
LIN {X 0,Y 506.133,Z 848.679,A -85,B 0,C 180,E1 22983.312,E2 22983.312} C_VEL
LIN {X 0,Y 503.052,Z 868.567,A -85,B 0,C 180,E1 22981.493,E2 22981.493} C_VEL
LIN {X 0,Y 500.267,Z 885.971,A -85,B 0,C 180,E1 22979.649,E2 22979.649} C_VEL
LIN {X 0,Y 497.521,Z 903.473,A -85,B 0,C 180,E1 22977.532,E2 22977.532} C_VEL
LIN {X 0,Y 495.271,Z 918.206,A -85,B 0,C 180,E1 22975.469,E2 22975.469} C_VEL
LIN {X 0,Y 493.099,Z 933.397,A -85,B 0,C 180,E1 22973.039,E2 22973.039} C_VEL
LIN {X 0,Y 491.491,Z 945.773,A -85,B 0,C 180,E1 22970.731,E2 22970.731} C_VEL
LIN {X 0,Y 490.173,Z 957.591,A -85,B 0,C 180,E1 22968.186,E2 22968.186} C_VEL
LIN {X 0,Y 489.254,Z 967.431,A -85,B 0,C 180,E1 22965.65,E2 22965.65} C_VEL
LIN {X 0,Y 488.666,Z 976.092,A -85,B 0,C 180,E1 22963.007,E2 22963.007} C_VEL
LIN {X 0,Y 488.356,Z 982.848,A -85,B 0,C 180,E1 22960.38,E2 22960.38} C_VEL
LIN {X 0,Y 488.246,Z 987.67,A -85,B 0,C 180,E1 22958.005,E2 22958.005} C_VEL
LIN {X 0,Y 488.235,Z 991.624,A -85,B 0,C 180,E1 22955.288,E2 22955.288} C_VEL
LIN {X 0,Y 488.278,Z 993.657,A -85,B 0,C 180,E1 22952.934,E2 22952.934} C_VEL
LIN {X 0,Y 488.31,Z 994.473,A -85,B 0,C 180,E1 22950.704,E2 22950.704} C_VEL
LIN {X 0,Y 488.328,Z 994.095,A -85,B 0,C 180,E1 22948.123,E2 22948.123} C_VEL
LIN {X 0,Y 488.308,Z 992.061,A -85,B 0,C 180,E1 22945.537,E2 22945.537} C_VEL
LIN {X 0,Y 488.303,Z 988.949,A -85,B 0,C 180,E1 22943.179,E2 22943.179} C_VEL
LIN {X 0,Y 488.368,Z 983.837,A -85,B 0,C 180,E1 22940.454,E2 22940.454} C_VEL
LIN {X 0,Y 488.591,Z 977.137,A -85,B 0,C 180,E1 22937.831,E2 22937.831} C_VEL
LIN {X 0,Y 489.01,Z 969.667,A -85,B 0,C 180,E1 22935.434,E2 22935.434} C_VEL
LIN {X 0,Y 489.822,Z 959.11,A -85,B 0,C 180,E1 22932.66,E2 22932.66} C_VEL
LIN {X 0,Y 490.822,Z 948.79,A -85,B 0,C 180,E1 22930.358,E2 22930.358} C_VEL
LIN {X 0,Y 492.431,Z 934.759,A -85,B 0,C 180,E1 22927.684,E2 22927.684} C_VEL
LIN {X 0,Y 494.254,Z 920.678,A -85,B 0,C 180,E1 22925.371,E2 22925.371} C_VEL
LIN {X 0,Y 496.543,Z 904.403,A -85,B 0,C 180,E1 22923.058,E2 22923.058} C_VEL
LIN {X 0,Y 499.003,Z 887.809,A -85,B 0,C 180,E1 22920.993,E2 22920.993} C_VEL
LIN {X 0,Y 501.911,Z 868.716,A -85,B 0,C 180,E1 22918.937,E2 22918.937} C_VEL
LIN {X 0,Y 504.876,Z 849.322,A -85,B 0,C 180,E1 22917.111,E2 22917.111} C_VEL
LIN {X 0,Y 507.891,Z 828.825,A -85,B 0,C 180,E1 22915.459,E2 22915.459} C_VEL
LIN {X 0,Y 510.965,Z 807.693,A -85,B 0,C 180,E1 22913.982,E2 22913.982} C_VEL
LIN {X 0,Y 513.725,Z 786.842,A -85,B 0,C 180,E1 22912.748,E2 22912.748} C_VEL
LIN {X 0,Y 516.513,Z 764.639,A -85,B 0,C 180,E1 22911.63,E2 22911.63} C_VEL
LIN {X 0,Y 518.91,Z 742.736,A -85,B 0,C 180,E1 22910.729,E2 22910.729} C_VEL
LIN {X 0,Y 521.22,Z 718.185,A -85,B 0,C 180,E1 22909.916,E2 22909.916} C_VEL
LIN {X 0,Y 523.123,Z 693.188,A -85,B 0,C 180,E1 22909.301,E2 22909.301} C_VEL
LIN {X 0,Y 528.462,Z 583.74,A -85,B 0,C 180,E1 22907.389,E2 22907.389} C_VEL
LIN {X 0,Y 533.562,Z 509.512,A -85,B 0,C 180,E1 22905.962,E2 22905.962} C_VEL
LIN {X 0,Y 540.211,Z 438.406,A -85,B 0,C 180,E1 22904.477,E2 22904.477} C_VEL
LIN {X 0,Y 548.593,Z 370.874,A -85,B 0,C 180,E1 22902.987,E2 22902.987} C_VEL
LIN {X 0,Y 550.864,Z 355.837,A -85,B 0,C 180,E1 22902.643,E2 22902.643} C_VEL
LIN {X 0,Y 553.527,Z 351.611,A -85,B 0,C 180,E1 22902.446,E2 22902.446} C_VEL
LIN {X 0,Y 557.392,Z 345.328,A -85,B 0,C 180,E1 22901.826,E2 22901.826} C_VEL
LIN {X 0,Y 547.265,Z 361.034,A -85,B 0,C 180,E1 22900.026,E2 22900.026} C_VEL
LIN {X 0,Y 541.273,Z 373.163,A -85,B 0,C 180,E1 22898.722,E2 22898.722} C_VEL
LIN {X 0,Y 538.529,Z 389.206,A -85,B 0,C 180,E1 22897.316,E2 22897.316} C_VEL
LIN {X 0,Y 536.557,Z 407.669,A -85,B 0,C 180,E1 22895.891,E2 22895.891} C_VEL
LIN {X 0,Y 535.061,Z 430.229,A -85,B 0,C 180,E1 22894.39,E2 22894.39} C_VEL
LIN {X 0,Y 533.805,Z 458.593,A -85,B 0,C 180,E1 22892.783,E2 22892.783} C_VEL
LIN {X 0,Y 532.714,Z 490.752,A -85,B 0,C 180,E1 22891.233,E2 22891.233} C_VEL
LIN {X 0,Y 531.971,Z 508.887,A -85,B 0,C 180,E1 22890.474,E2 22890.474} C_VEL
LIN {X 0,Y 519.156,Z 616.895,A -85,B 0,C 180,E1 22887.652,E2 22887.652} C_VEL
LIN {X 0,Y 512.023,Z 690.774,A -85,B 0,C 180,E1 22885.696,E2 22885.696} C_VEL
LIN {X 0,Y 509.623,Z 714.531,A -85,B 0,C 180,E1 22884.858,E2 22884.858} C_VEL
LIN {X 0,Y 507.126,Z 738.308,A -85,B 0,C 180,E1 22883.779,E2 22883.779} C_VEL
LIN {X 0,Y 504.819,Z 759.265,A -85,B 0,C 180,E1 22882.598,E2 22882.598} C_VEL
LIN {X 0,Y 502.66,Z 778.514,A -85,B 0,C 180,E1 22881.286,E2 22881.286} C_VEL
LIN {X 0,Y 500.462,Z 797.298,A -85,B 0,C 180,E1 22879.734,E2 22879.734} C_VEL
LIN {X 0,Y 498.615,Z 812.524,A -85,B 0,C 180,E1 22878.23,E2 22878.23} C_VEL
LIN {X 0,Y 496.895,Z 826.413,A -85,B 0,C 180,E1 22876.603,E2 22876.603} C_VEL
LIN {X 0,Y 495.3,Z 838.799,A -85,B 0,C 180,E1 22874.856,E2 22874.856} C_VEL
LIN {X 0,Y 493.962,Z 849.119,A -85,B 0,C 180,E1 22873.104,E2 22873.104} C_VEL
LIN {X 0,Y 492.693,Z 858.533,A -85,B 0,C 180,E1 22871.116,E2 22871.116} C_VEL
LIN {X 0,Y 491.695,Z 865.896,A -85,B 0,C 180,E1 22869.127,E2 22869.127} C_VEL
LIN {X 0,Y 490.924,Z 871.352,A -85,B 0,C 180,E1 22867.137,E2 22867.137} C_VEL
LIN {X 0,Y 490.35,Z 875.114,A -85,B 0,C 180,E1 22865.148,E2 22865.148} C_VEL
LIN {X 0,Y 489.918,Z 877.331,A -85,B 0,C 180,E1 22863.042,E2 22863.042} C_VEL
LIN {X 0,Y 489.633,Z 877.765,A -85,B 0,C 180,E1 22860.936,E2 22860.936} C_VEL
LIN {X 0,Y 489.477,Z 876.465,A -85,B 0,C 180,E1 22858.829,E2 22858.829} C_VEL
LIN {X 0,Y 489.433,Z 873.448,A -85,B 0,C 180,E1 22856.721,E2 22856.721} C_VEL
LIN {X 0,Y 489.52,Z 868.653,A -85,B 0,C 180,E1 22854.609,E2 22854.609} C_VEL
LIN {X 0,Y 489.765,Z 862.002,A -85,B 0,C 180,E1 22852.492,E2 22852.492} C_VEL
LIN {X 0,Y 490.208,Z 853.338,A -85,B 0,C 180,E1 22850.372,E2 22850.372} C_VEL
LIN {X 0,Y 490.861,Z 843.095,A -85,B 0,C 180,E1 22848.366,E2 22848.366} C_VEL
LIN {X 0,Y 491.709,Z 831.353,A -85,B 0,C 180,E1 22846.476,E2 22846.476} C_VEL
LIN {X 0,Y 492.741,Z 818.133,A -85,B 0,C 180,E1 22844.704,E2 22844.704} C_VEL
LIN {X 0,Y 493.933,Z 803.449,A -85,B 0,C 180,E1 22843.052,E2 22843.052} C_VEL
LIN {X 0,Y 495.268,Z 787.239,A -85,B 0,C 180,E1 22841.52,E2 22841.52} C_VEL
LIN {X 0,Y 496.696,Z 769.35,A -85,B 0,C 180,E1 22840.11,E2 22840.11} C_VEL
LIN {X 0,Y 498.155,Z 750.407,A -85,B 0,C 180,E1 22838.882,E2 22838.882} C_VEL
LIN {X 0,Y 499.578,Z 730.331,A -85,B 0,C 180,E1 22837.835,E2 22837.835} C_VEL
LIN {X 0,Y 500.861,Z 709.536,A -85,B 0,C 180,E1 22836.985,E2 22836.985} C_VEL
LIN {X 0,Y 501.993,Z 688.039,A -85,B 0,C 180,E1 22836.333,E2 22836.333} C_VEL
LIN {X 0,Y 503.092,Z 659.124,A -85,B 0,C 180,E1 22835.742,E2 22835.742} C_VEL
LIN {X 0,Y 509.188,Z 498.647,A -85,B 0,C 180,E1 22832.72,E2 22832.72} C_VEL
LIN {X 0,Y 504.307,Z 446.424,A -85,B 0,C 180,E1 22831.294,E2 22831.294} C_VEL
LIN {X 0,Y 508.678,Z 393.244,A -85,B 0,C 180,E1 22827.412,E2 22827.412} C_VEL
LIN {X 0,Y 513.168,Z 344.374,A -85,B 0,C 180,E1 22823.815,E2 22823.815} C_VEL
LIN {X 0,Y 518.183,Z 294.693,A -85,B 0,C 180,E1 22820.125,E2 22820.125} C_VEL
LIN {X 0,Y 510.877,Z 274.648,A -85,B 0,C 180,E1 22817.831,E2 22817.831} C_VEL
LIN {X 0,Y 507.832,Z 266.752,A -85,B 0,C 180,E1 22816.865,E2 22816.865} C_VEL
LIN {X 0,Y 510.169,Z 267.426,A -85,B 0,C 180,E1 22816.533,E2 22816.533} C_VEL
LIN {X 0,Y 513.169,Z 267.803,A -85,B 0,C 180,E1 22816.149,E2 22816.149} C_VEL
LIN {X 0,Y 521.029,Z 285.994,A -85,B 0,C 180,E1 22813.851,E2 22813.851} C_VEL
LIN {X 0,Y 528.966,Z 307.024,A -85,B 0,C 180,E1 22811.371,E2 22811.371} C_VEL
LIN {X 0,Y 530.034,Z 310.339,A -85,B 0,C 180,E1 22811.01,E2 22811.01} C_VEL
LIN {X 0,Y 529.565,Z 353.244,A -85,B 0,C 180,E1 22808.061,E2 22808.061} C_VEL
LIN {X 0,Y 529.287,Z 356.557,A -85,B 0,C 180,E1 22807.877,E2 22807.877} C_VEL
LIN {X 0,Y 526.333,Z 370.726,A -85,B 0,C 180,E1 22807.349,E2 22807.349} C_VEL
LIN {X 0,Y 523.463,Z 455.536,A -85,B 0,C 180,E1 22806.066,E2 22806.066} C_VEL
LIN {X 0,Y 522.35,Z 463.2,A -85,B 0,C 180,E1 22806.004,E2 22806.004} C_VEL
LIN {X 0,Y 516.416,Z 483.598,A -85,B 0,C 180,E1 22806.075,E2 22806.075} C_VEL
LIN {X 0,Y 515.507,Z 490.169,A -85,B 0,C 180,E1 22806.009,E2 22806.009} C_VEL
LIN {X 0,Y 511.4,Z 563.586,A -85,B 0,C 180,E1 22804.596,E2 22804.596} C_VEL
LIN {X 0,Y 507.033,Z 634.713,A -85,B 0,C 180,E1 22803.026,E2 22803.026} C_VEL
LIN {X 0,Y 505.734,Z 660.074,A -85,B 0,C 180,E1 22802.318,E2 22802.318} C_VEL
LIN {X 0,Y 504.192,Z 681.993,A -85,B 0,C 180,E1 22801.487,E2 22801.487} C_VEL
LIN {X 0,Y 502.295,Z 703.148,A -85,B 0,C 180,E1 22800.463,E2 22800.463} C_VEL
LIN {X 0,Y 500.238,Z 722.454,A -85,B 0,C 180,E1 22799.322,E2 22799.322} C_VEL
LIN {X 0,Y 497.916,Z 741.578,A -85,B 0,C 180,E1 22797.963,E2 22797.963} C_VEL
LIN {X 0,Y 495.319,Z 760.847,A -85,B 0,C 180,E1 22796.324,E2 22796.324} C_VEL
LIN {X 0,Y 492.74,Z 778.685,A -85,B 0,C 180,E1 22794.518,E2 22794.518} C_VEL
LIN {X 0,Y 490.405,Z 794.185,A -85,B 0,C 180,E1 22792.666,E2 22792.666} C_VEL
LIN {X 0,Y 488.202,Z 808.74,A -85,B 0,C 180,E1 22790.627,E2 22790.627} C_VEL
LIN {X 0,Y 486.252,Z 821.862,A -85,B 0,C 180,E1 22788.462,E2 22788.462} C_VEL
LIN {X 0,Y 484.599,Z 833.539,A -85,B 0,C 180,E1 22786.174,E2 22786.174} C_VEL
LIN {X 0,Y 483.344,Z 843.311,A -85,B 0,C 180,E1 22783.885,E2 22783.885} C_VEL
LIN {X 0,Y 482.33,Z 852.187,A -85,B 0,C 180,E1 22781.318,E2 22781.318} C_VEL
LIN {X 0,Y 481.668,Z 858.843,A -85,B 0,C 180,E1 22778.837,E2 22778.837} C_VEL
LIN {X 0,Y 481.264,Z 863.864,A -85,B 0,C 180,E1 22776.322,E2 22776.322} C_VEL
LIN {X 0,Y 481.043,Z 867.331,A -85,B 0,C 180,E1 22773.695,E2 22773.695} C_VEL
LIN {X 0,Y 480.959,Z 868.969,A -85,B 0,C 180,E1 22771.31,E2 22771.31} C_VEL
LIN {X 0,Y 480.949,Z 869.03,A -85,B 0,C 180,E1 22768.928,E2 22768.928} C_VEL
LIN {X 0,Y 481.028,Z 867.529,A -85,B 0,C 180,E1 22766.425,E2 22766.425} C_VEL
LIN {X 0,Y 481.221,Z 864.628,A -85,B 0,C 180,E1 22764.037,E2 22764.037} C_VEL
LIN {X 0,Y 481.579,Z 859.91,A -85,B 0,C 180,E1 22761.523,E2 22761.523} C_VEL
LIN {X 0,Y 482.151,Z 853.726,A -85,B 0,C 180,E1 22759.122,E2 22759.122} C_VEL
LIN {X 0,Y 483.082,Z 845.426,A -85,B 0,C 180,E1 22756.596,E2 22756.596} C_VEL
LIN {X 0,Y 484.352,Z 835.486,A -85,B 0,C 180,E1 22754.157,E2 22754.157} C_VEL
LIN {X 0,Y 485.91,Z 824.386,A -85,B 0,C 180,E1 22751.897,E2 22751.897} C_VEL
LIN {X 0,Y 487.781,Z 811.751,A -85,B 0,C 180,E1 22749.731,E2 22749.731} C_VEL
LIN {X 0,Y 490.049,Z 796.719,A -85,B 0,C 180,E1 22747.563,E2 22747.563} C_VEL
LIN {X 0,Y 492.448,Z 780.749,A -85,B 0,C 180,E1 22745.618,E2 22745.618} C_VEL
LIN {X 0,Y 494.892,Z 763.848,A -85,B 0,C 180,E1 22743.867,E2 22743.867} C_VEL
LIN {X 0,Y 497.303,Z 746.331,A -85,B 0,C 180,E1 22742.325,E2 22742.325} C_VEL
LIN {X 0,Y 499.687,Z 727.281,A -85,B 0,C 180,E1 22740.906,E2 22740.906} C_VEL
LIN {X 0,Y 501.796,Z 708.408,A -85,B 0,C 180,E1 22739.726,E2 22739.726} C_VEL
LIN {X 0,Y 503.782,Z 687.768,A -85,B 0,C 180,E1 22738.667,E2 22738.667} C_VEL
LIN {X 0,Y 505.438,Z 665.945,A -85,B 0,C 180,E1 22737.782,E2 22737.782} C_VEL
LIN {X 0,Y 506.645,Z 643.674,A -85,B 0,C 180,E1 22737.101,E2 22737.101} C_VEL
LIN {X 0,Y 509.577,Z 593.204,A -85,B 0,C 180,E1 22735.934,E2 22735.934} C_VEL
LIN {X 0,Y 513.995,Z 519.954,A -85,B 0,C 180,E1 22734.446,E2 22734.446} C_VEL
LIN {X 0,Y 517.243,Z 453.278,A -85,B 0,C 180,E1 22733.265,E2 22733.265} C_VEL
LIN {X 0,Y 520.245,Z 371.682,A -85,B 0,C 180,E1 22732,E2 22732} C_VEL
LIN {X 0,Y 523.543,Z 356.929,A -85,B 0,C 180,E1 22731.423,E2 22731.423} C_VEL
LIN {X 0,Y 523.906,Z 318.049,A -85,B 0,C 180,E1 22728.761,E2 22728.761} C_VEL
LIN {X 0,Y 523.867,Z 313.625,A -85,B 0,C 180,E1 22728.435,E2 22728.435} C_VEL
LIN {X 0,Y 516.028,Z 292.446,A -85,B 0,C 180,E1 22725.923,E2 22725.923} C_VEL
LIN {X 0,Y 507.554,Z 272.816,A -85,B 0,C 180,E1 22723.436,E2 22723.436} C_VEL
LIN {X 0,Y 499.437,Z 256.421,A -85,B 0,C 180,E1 22721.17,E2 22721.17} C_VEL
LIN {X 0,Y 492.888,Z 244.232,A -85,B 0,C 180,E1 22719.384,E2 22719.384} C_VEL
LIN {X 0,Y 487.544,Z 235.054,A -85,B 0,C 180,E1 22717.971,E2 22717.971} C_VEL
LIN {X 0,Y 485.446,Z 231.607,A -85,B 0,C 180,E1 22717.418,E2 22717.418} C_VEL
LIN {X 0,Y 484.643,Z 230.133,A -85,B 0,C 180,E1 22717.193,E2 22717.193} C_VEL
LIN {X 0,Y 482.495,Z 227.01,A -85,B 0,C 180,E1 22716.644,E2 22716.644} C_VEL
LIN {X 0,Y 482.043,Z 225.162,A -85,B 0,C 180,E1 22716.407,E2 22716.407} C_VEL
LIN {X 0,Y 482.035,Z 225.158,A -85,B 0,C 180,E1 22712.779,E2 22712.779} C_VEL
LIN {X 0,Y 482.048,Z 225.158,A -85,B 0,C 180,E1 22709.16,E2 22709.16} C_VEL
LIN {X 0,Y 482.049,Z 225.181,A -85,B 0,C 180,E1 22705.538,E2 22705.538} C_VEL
LIN {X 0,Y 482.044,Z 225.166,A -85,B 0,C 180,E1 22701.924,E2 22701.924} C_VEL
LIN {X 0,Y 482.045,Z 225.143,A -85,B 0,C 180,E1 22698.378,E2 22698.378} C_VEL
LIN {X 0,Y 482.048,Z 225.182,A -85,B 0,C 180,E1 22694.782,E2 22694.782} C_VEL
LIN {X 0,Y 482.045,Z 225.151,A -85,B 0,C 180,E1 22691.123,E2 22691.123} C_VEL
LIN {X 0,Y 482.033,Z 225.163,A -85,B 0,C 180,E1 22687.509,E2 22687.509} C_VEL
LIN {X 0,Y 482.037,Z 225.172,A -85,B 0,C 180,E1 22683.854,E2 22683.854} C_VEL
LIN {X 0,Y 482.053,Z 225.141,A -85,B 0,C 180,E1 22680.238,E2 22680.238} C_VEL
LIN {X 0,Y 482.05,Z 225.182,A -85,B 0,C 180,E1 22676.551,E2 22676.551} C_VEL
LIN {X 0,Y 482.056,Z 225.134,A -85,B 0,C 180,E1 22672.851,E2 22672.851} C_VEL
LIN {X 0,Y 482.032,Z 225.185,A -85,B 0,C 180,E1 22669.24,E2 22669.24} C_VEL
LIN {X 0,Y 482.025,Z 225.184,A -85,B 0,C 180,E1 22665.586,E2 22665.586} C_VEL
LIN {X 0,Y 482.04,Z 225.178,A -85,B 0,C 180,E1 22661.997,E2 22661.997} C_VEL
LIN {X 0,Y 482.059,Z 225.174,A -85,B 0,C 180,E1 22658.461,E2 22658.461} C_VEL
LIN {X 0,Y 482.04,Z 225.184,A -85,B 0,C 180,E1 22654.835,E2 22654.835} C_VEL
LIN {X 0,Y 482.032,Z 225.293,A -85,B 0,C 180,E1 22651.485,E2 22651.485} C_VEL
LIN {X 0,Y 483.413,Z 228.767,A -85,B 0,C 180,E1 22650.917,E2 22650.917} C_VEL
LIN {X 0,Y 484.613,Z 230.742,A -85,B 0,C 180,E1 22650.54,E2 22650.54} C_VEL
LIN {X 0,Y 491.59,Z 244.301,A -85,B 0,C 180,E1 22648.21,E2 22648.21} C_VEL
LIN {X 0,Y 501.162,Z 263.07,A -85,B 0,C 180,E1 22645.207,E2 22645.207} C_VEL
LIN {X 0,Y 510.817,Z 282.52,A -85,B 0,C 180,E1 22642.358,E2 22642.358} C_VEL
LIN {X 0,Y 521.719,Z 305.144,A -85,B 0,C 180,E1 22639.336,E2 22639.336} C_VEL
LIN {X 0,Y 527.639,Z 317.579,A -85,B 0,C 180,E1 22637.831,E2 22637.831} C_VEL
LIN {X 0,Y 528.388,Z 319.377,A -85,B 0,C 180,E1 22637.728,E2 22637.728} C_VEL
LIN {X 0,Y 530.976,Z 346.541,A -85,B 0,C 180,E1 22636.943,E2 22636.943} C_VEL
LIN {X 0,Y 520.798,Z 584.167,A -85,B 0,C 180,E1 22633.035,E2 22633.035} C_VEL
LIN {X 0,Y 516.743,Z 692.909,A -85,B 0,C 180,E1 22631.271,E2 22631.271} C_VEL
LIN {X 0,Y 514.996,Z 717.542,A -85,B 0,C 180,E1 22630.688,E2 22630.688} C_VEL
LIN {X 0,Y 512.9,Z 741.527,A -85,B 0,C 180,E1 22629.935,E2 22629.935} C_VEL
LIN {X 0,Y 510.48,Z 763.973,A -85,B 0,C 180,E1 22629.03,E2 22629.03} C_VEL
LIN {X 0,Y 507.695,Z 786.913,A -85,B 0,C 180,E1 22627.914,E2 22627.914} C_VEL
LIN {X 0,Y 504.938,Z 807.104,A -85,B 0,C 180,E1 22626.729,E2 22626.729} C_VEL
LIN {X 0,Y 501.736,Z 828.946,A -85,B 0,C 180,E1 22625.235,E2 22625.235} C_VEL
LIN {X 0,Y 498.725,Z 848.133,A -85,B 0,C 180,E1 22623.692,E2 22623.692} C_VEL
LIN {X 0,Y 495.535,Z 868.127,A -85,B 0,C 180,E1 22621.843,E2 22621.843} C_VEL
LIN {X 0,Y 492.721,Z 885.167,A -85,B 0,C 180,E1 22620.015,E2 22620.015} C_VEL
LIN {X 0,Y 489.866,Z 902.698,A -85,B 0,C 180,E1 22617.867,E2 22617.867} C_VEL
LIN {X 0,Y 487.535,Z 917.493,A -85,B 0,C 180,E1 22615.772,E2 22615.772} C_VEL
LIN {X 0,Y 485.38,Z 932.046,A -85,B 0,C 180,E1 22613.427,E2 22613.427} C_VEL
LIN {X 0,Y 483.617,Z 945.097,A -85,B 0,C 180,E1 22610.958,E2 22610.958} C_VEL
LIN {X 0,Y 482.24,Z 956.932,A -85,B 0,C 180,E1 22608.37,E2 22608.37} C_VEL
LIN {X 0,Y 481.315,Z 966.481,A -85,B 0,C 180,E1 22605.878,E2 22605.878} C_VEL
LIN {X 0,Y 480.711,Z 975.059,A -85,B 0,C 180,E1 22603.227,E2 22603.227} C_VEL
LIN {X 0,Y 480.38,Z 982.148,A -85,B 0,C 180,E1 22600.433,E2 22600.433} C_VEL
LIN {X 0,Y 480.277,Z 986.95,A -85,B 0,C 180,E1 22598.018,E2 22598.018} C_VEL
LIN {X 0,Y 480.276,Z 990.842,A -85,B 0,C 180,E1 22595.256,E2 22595.256} C_VEL
LIN {X 0,Y 480.325,Z 992.832,A -85,B 0,C 180,E1 22592.864,E2 22592.864} C_VEL
LIN {X 0,Y 480.359,Z 993.6,A -85,B 0,C 180,E1 22590.596,E2 22590.596} C_VEL
LIN {X 0,Y 480.373,Z 993.062,A -85,B 0,C 180,E1 22587.853,E2 22587.853} C_VEL
LIN {X 0,Y 480.341,Z 991.019,A -85,B 0,C 180,E1 22585.343,E2 22585.343} C_VEL
LIN {X 0,Y 480.333,Z 988.012,A -85,B 0,C 180,E1 22583.065,E2 22583.065} C_VEL
LIN {X 0,Y 480.399,Z 982.868,A -85,B 0,C 180,E1 22580.294,E2 22580.294} C_VEL
LIN {X 0,Y 480.63,Z 976.14,A -85,B 0,C 180,E1 22577.627,E2 22577.627} C_VEL
LIN {X 0,Y 481.098,Z 968.23,A -85,B 0,C 180,E1 22575.065,E2 22575.065} C_VEL
LIN {X 0,Y 481.928,Z 958.026,A -85,B 0,C 180,E1 22572.367,E2 22572.367} C_VEL
LIN {X 0,Y 483.045,Z 947.101,A -85,B 0,C 180,E1 22569.903,E2 22569.903} C_VEL
LIN {X 0,Y 484.741,Z 933.138,A -85,B 0,C 180,E1 22567.227,E2 22567.227} C_VEL
LIN {X 0,Y 486.733,Z 918.717,A -85,B 0,C 180,E1 22564.834,E2 22564.834} C_VEL
LIN {X 0,Y 489.164,Z 902.254,A -85,B 0,C 180,E1 22562.486,E2 22562.486} C_VEL
LIN {X 0,Y 491.937,Z 884.819,A -85,B 0,C 180,E1 22560.306,E2 22560.306} C_VEL
LIN {X 0,Y 494.968,Z 865.802,A -85,B 0,C 180,E1 22558.263,E2 22558.263} C_VEL
LIN {X 0,Y 498.219,Z 845.5,A -85,B 0,C 180,E1 22556.364,E2 22556.364} C_VEL
LIN {X 0,Y 501.361,Z 825.535,A -85,B 0,C 180,E1 22554.757,E2 22554.757} C_VEL
LIN {X 0,Y 504.856,Z 802.069,A -85,B 0,C 180,E1 22553.144,E2 22553.144} C_VEL
LIN {X 0,Y 508.054,Z 779.456,A -85,B 0,C 180,E1 22551.831,E2 22551.831} C_VEL
LIN {X 0,Y 511.015,Z 755.84,A -85,B 0,C 180,E1 22550.71,E2 22550.71} C_VEL
LIN {X 0,Y 513.846,Z 730.482,A -85,B 0,C 180,E1 22549.741,E2 22549.741} C_VEL
LIN {X 0,Y 516.054,Z 707.13,A -85,B 0,C 180,E1 22549.047,E2 22549.047} C_VEL
LIN {X 0,Y 517.709,Z 682.779,A -85,B 0,C 180,E1 22548.52,E2 22548.52} C_VEL
LIN {X 0,Y 522.492,Z 593.531,A -85,B 0,C 180,E1 22546.921,E2 22546.921} C_VEL
LIN {X 0,Y 527.819,Z 522.285,A -85,B 0,C 180,E1 22545.518,E2 22545.518} C_VEL
LIN {X 0,Y 534.576,Z 454.884,A -85,B 0,C 180,E1 22544.075,E2 22544.075} C_VEL
LIN {X 0,Y 542.768,Z 392.347,A -85,B 0,C 180,E1 22542.675,E2 22542.675} C_VEL
LIN {X 0,Y 548.127,Z 358.958,A -85,B 0,C 180,E1 22541.903,E2 22541.903} C_VEL
LIN {X 0,Y 550.284,Z 355.693,A -85,B 0,C 180,E1 22541.755,E2 22541.755} C_VEL
LIN {X 0,Y 544.284,Z 365.012,A -85,B 0,C 180,E1 22540.688,E2 22540.688} C_VEL
LIN {X 0,Y 539.398,Z 380.968,A -85,B 0,C 180,E1 22539.121,E2 22539.121} C_VEL
LIN {X 0,Y 536.467,Z 395.147,A -85,B 0,C 180,E1 22537.873,E2 22537.873} C_VEL
LIN {X 0,Y 533.779,Z 414.563,A -85,B 0,C 180,E1 22536.37,E2 22536.37} C_VEL
LIN {X 0,Y 531.595,Z 437.999,A -85,B 0,C 180,E1 22534.827,E2 22534.827} C_VEL
LIN {X 0,Y 529.823,Z 465.534,A -85,B 0,C 180,E1 22533.263,E2 22533.263} C_VEL
LIN {X 0,Y 528.165,Z 497.407,A -85,B 0,C 180,E1 22531.716,E2 22531.716} C_VEL
LIN {X 0,Y 527.364,Z 510.645,A -85,B 0,C 180,E1 22531.16,E2 22531.16} C_VEL
LIN {X 0,Y 513.633,Z 618.773,A -85,B 0,C 180,E1 22528.272,E2 22528.272} C_VEL
LIN {X 0,Y 505.897,Z 692.84,A -85,B 0,C 180,E1 22526.245,E2 22526.245} C_VEL
LIN {X 0,Y 503.288,Z 716.231,A -85,B 0,C 180,E1 22525.381,E2 22525.381} C_VEL
LIN {X 0,Y 500.643,Z 739.505,A -85,B 0,C 180,E1 22524.295,E2 22524.295} C_VEL
LIN {X 0,Y 497.962,Z 761.93,A -85,B 0,C 180,E1 22522.989,E2 22522.989} C_VEL
LIN {X 0,Y 495.654,Z 780.628,A -85,B 0,C 180,E1 22521.664,E2 22521.664} C_VEL
LIN {X 0,Y 493.5,Z 797.932,A -85,B 0,C 180,E1 22520.21,E2 22520.21} C_VEL
LIN {X 0,Y 491.299,Z 814.753,A -85,B 0,C 180,E1 22518.511,E2 22518.511} C_VEL
LIN {X 0,Y 489.46,Z 828.363,A -85,B 0,C 180,E1 22516.863,E2 22516.863} C_VEL
LIN {X 0,Y 487.778,Z 840.637,A -85,B 0,C 180,E1 22515.09,E2 22515.09} C_VEL
LIN {X 0,Y 486.254,Z 851.38,A -85,B 0,C 180,E1 22513.194,E2 22513.194} C_VEL
LIN {X 0,Y 485,Z 860.123,A -85,B 0,C 180,E1 22511.295,E2 22511.295} C_VEL
LIN {X 0,Y 483.928,Z 867.372,A -85,B 0,C 180,E1 22509.274,E2 22509.274} C_VEL
LIN {X 0,Y 483.068,Z 873.043,A -85,B 0,C 180,E1 22507.134,E2 22507.134} C_VEL
LIN {X 0,Y 482.428,Z 876.766,A -85,B 0,C 180,E1 22504.994,E2 22504.994} C_VEL
LIN {X 0,Y 481.978,Z 878.679,A -85,B 0,C 180,E1 22502.854,E2 22502.854} C_VEL
LIN {X 0,Y 481.691,Z 878.819,A -85,B 0,C 180,E1 22500.714,E2 22500.714} C_VEL
LIN {X 0,Y 481.53,Z 877.212,A -85,B 0,C 180,E1 22498.572,E2 22498.572} C_VEL
LIN {X 0,Y 481.494,Z 873.875,A -85,B 0,C 180,E1 22496.428,E2 22496.428} C_VEL
LIN {X 0,Y 481.605,Z 868.768,A -85,B 0,C 180,E1 22494.281,E2 22494.281} C_VEL
LIN {X 0,Y 481.881,Z 861.783,A -85,B 0,C 180,E1 22492.129,E2 22492.129} C_VEL
LIN {X 0,Y 482.339,Z 853.305,A -85,B 0,C 180,E1 22490.092,E2 22490.092} C_VEL
LIN {X 0,Y 483.039,Z 842.79,A -85,B 0,C 180,E1 22488.053,E2 22488.053} C_VEL
LIN {X 0,Y 483.945,Z 830.754,A -85,B 0,C 180,E1 22486.133,E2 22486.133} C_VEL
LIN {X 0,Y 485.074,Z 816.864,A -85,B 0,C 180,E1 22484.288,E2 22484.288} C_VEL
LIN {X 0,Y 486.362,Z 801.625,A -85,B 0,C 180,E1 22482.595,E2 22482.595} C_VEL
LIN {X 0,Y 487.79,Z 784.779,A -85,B 0,C 180,E1 22481.032,E2 22481.032} C_VEL
LIN {X 0,Y 489.22,Z 767.155,A -85,B 0,C 180,E1 22479.668,E2 22479.668} C_VEL
LIN {X 0,Y 490.684,Z 748.607,A -85,B 0,C 180,E1 22478.482,E2 22478.482} C_VEL
LIN {X 0,Y 492.088,Z 729.343,A -85,B 0,C 180,E1 22477.479,E2 22477.479} C_VEL
LIN {X 0,Y 493.436,Z 708.088,A -85,B 0,C 180,E1 22476.613,E2 22476.613} C_VEL
LIN {X 0,Y 494.621,Z 686.149,A -85,B 0,C 180,E1 22475.954,E2 22475.954} C_VEL
LIN {X 0,Y 496.191,Z 644.603,A -85,B 0,C 180,E1 22475.12,E2 22475.12} C_VEL
LIN {X 0,Y 501.976,Z 499.387,A -85,B 0,C 180,E1 22472.329,E2 22472.329} C_VEL
LIN {X 0,Y 497.08,Z 445.289,A -85,B 0,C 180,E1 22470.81,E2 22470.81} C_VEL
LIN {X 0,Y 501.552,Z 393.19,A -85,B 0,C 180,E1 22466.958,E2 22466.958} C_VEL
LIN {X 0,Y 506.339,Z 343.384,A -85,B 0,C 180,E1 22463.248,E2 22463.248} C_VEL
LIN {X 0,Y 511.134,Z 297.518,A -85,B 0,C 180,E1 22459.801,E2 22459.801} C_VEL
LIN {X 0,Y 502.711,Z 274.81,A -85,B 0,C 180,E1 22457.138,E2 22457.138} C_VEL
LIN {X 0,Y 502.414,Z 273.908,A -85,B 0,C 180,E1 22457.007,E2 22457.007} C_VEL
LIN {X 0,Y 504.462,Z 274.528,A -85,B 0,C 180,E1 22456.701,E2 22456.701} C_VEL
LIN {X 0,Y 508.475,Z 274.849,A -85,B 0,C 180,E1 22456.194,E2 22456.194} C_VEL
LIN {X 0,Y 516.549,Z 293.957,A -85,B 0,C 180,E1 22453.778,E2 22453.778} C_VEL
LIN {X 0,Y 523.91,Z 313.859,A -85,B 0,C 180,E1 22451.432,E2 22451.432} C_VEL
LIN {X 0,Y 523.449,Z 356.947,A -85,B 0,C 180,E1 22448.472,E2 22448.472} C_VEL
LIN {X 0,Y 519.968,Z 373.528,A -85,B 0,C 180,E1 22447.853,E2 22447.853} C_VEL
LIN {X 0,Y 516.931,Z 459.567,A -85,B 0,C 180,E1 22446.537,E2 22446.537} C_VEL
LIN {X 0,Y 515.507,Z 490.169,A -85,B 0,C 180,E1 22446.009,E2 22446.009} C_VEL
LIN {X 0,Y 514.345,Z 497.819,A -85,B 0,C 180,E1 22445.938,E2 22445.938} C_VEL
LIN {X 0,Y 508.267,Z 518.177,A -85,B 0,C 180,E1 22445.983,E2 22445.983} C_VEL
LIN {X 0,Y 507.289,Z 524.733,A -85,B 0,C 180,E1 22445.908,E2 22445.908} C_VEL
LIN {X 0,Y 502.493,Z 600.764,A -85,B 0,C 180,E1 22444.326,E2 22444.326} C_VEL
LIN {X 0,Y 499.772,Z 646.534,A -85,B 0,C 180,E1 22443.23,E2 22443.23} C_VEL
LIN {X 0,Y 498.54,Z 668.142,A -85,B 0,C 180,E1 22442.549,E2 22442.549} C_VEL
LIN {X 0,Y 496.811,Z 689.973,A -85,B 0,C 180,E1 22441.642,E2 22441.642} C_VEL
LIN {X 0,Y 494.724,Z 710.777,A -85,B 0,C 180,E1 22440.551,E2 22440.551} C_VEL
LIN {X 0,Y 492.444,Z 730.313,A -85,B 0,C 180,E1 22439.297,E2 22439.297} C_VEL
LIN {X 0,Y 489.968,Z 749.027,A -85,B 0,C 180,E1 22437.861,E2 22437.861} C_VEL
LIN {X 0,Y 487.302,Z 767.508,A -85,B 0,C 180,E1 22436.178,E2 22436.178} C_VEL
LIN {X 0,Y 484.655,Z 784.843,A -85,B 0,C 180,E1 22434.305,E2 22434.305} C_VEL
LIN {X 0,Y 482.176,Z 800.537,A -85,B 0,C 180,E1 22432.302,E2 22432.302} C_VEL
LIN {X 0,Y 479.994,Z 814.356,A -85,B 0,C 180,E1 22430.231,E2 22430.231} C_VEL
LIN {X 0,Y 478.09,Z 826.817,A -85,B 0,C 180,E1 22428.031,E2 22428.031} C_VEL
LIN {X 0,Y 476.381,Z 838.536,A -85,B 0,C 180,E1 22425.546,E2 22425.546} C_VEL
LIN {X 0,Y 475.075,Z 848.28,A -85,B 0,C 180,E1 22423.015,E2 22423.015} C_VEL
LIN {X 0,Y 474.193,Z 855.818,A -85,B 0,C 180,E1 22420.571,E2 22420.571} C_VEL
LIN {X 0,Y 473.59,Z 861.948,A -85,B 0,C 180,E1 22418.01,E2 22418.01} C_VEL
LIN {X 0,Y 473.251,Z 866.357,A -85,B 0,C 180,E1 22415.456,E2 22415.456} C_VEL
LIN {X 0,Y 473.077,Z 869.113,A -85,B 0,C 180,E1 22412.908,E2 22412.908} C_VEL
LIN {X 0,Y 473.009,Z 870.147,A -85,B 0,C 180,E1 22410.363,E2 22410.363} C_VEL
LIN {X 0,Y 473.046,Z 869.578,A -85,B 0,C 180,E1 22407.82,E2 22407.82} C_VEL
LIN {X 0,Y 473.186,Z 867.412,A -85,B 0,C 180,E1 22405.273,E2 22405.273} C_VEL
LIN {X 0,Y 473.468,Z 863.613,A -85,B 0,C 180,E1 22402.721,E2 22402.721} C_VEL
LIN {X 0,Y 473.968,Z 858.017,A -85,B 0,C 180,E1 22400.161,E2 22400.161} C_VEL
LIN {X 0,Y 474.756,Z 851.005,A -85,B 0,C 180,E1 22397.718,E2 22397.718} C_VEL
LIN {X 0,Y 475.921,Z 841.751,A -85,B 0,C 180,E1 22395.148,E2 22395.148} C_VEL
LIN {X 0,Y 477.437,Z 831.152,A -85,B 0,C 180,E1 22392.746,E2 22392.746} C_VEL
LIN {X 0,Y 479.248,Z 819.296,A -85,B 0,C 180,E1 22390.499,E2 22390.499} C_VEL
LIN {X 0,Y 481.426,Z 805.537,A -85,B 0,C 180,E1 22388.303,E2 22388.303} C_VEL
LIN {X 0,Y 483.853,Z 790.18,A -85,B 0,C 180,E1 22386.236,E2 22386.236} C_VEL
LIN {X 0,Y 486.381,Z 773.879,A -85,B 0,C 180,E1 22384.375,E2 22384.375} C_VEL
LIN {X 0,Y 488.969,Z 756.338,A -85,B 0,C 180,E1 22382.672,E2 22382.672} C_VEL
LIN {X 0,Y 491.47,Z 738.084,A -85,B 0,C 180,E1 22381.173,E2 22381.173} C_VEL
LIN {X 0,Y 493.925,Z 718.094,A -85,B 0,C 180,E1 22379.798,E2 22379.798} C_VEL
LIN {X 0,Y 496.061,Z 698.144,A -85,B 0,C 180,E1 22378.665,E2 22378.665} C_VEL
LIN {X 0,Y 497.882,Z 677.418,A -85,B 0,C 180,E1 22377.71,E2 22377.71} C_VEL
LIN {X 0,Y 499.402,Z 655.167,A -85,B 0,C 180,E1 22376.918,E2 22376.918} C_VEL
LIN {X 0,Y 501.293,Z 619.373,A -85,B 0,C 180,E1 22376.001,E2 22376.001} C_VEL
LIN {X 0,Y 506.162,Z 544.365,A -85,B 0,C 180,E1 22374.382,E2 22374.382} C_VEL
LIN {X 0,Y 509.917,Z 475.713,A -85,B 0,C 180,E1 22373.093,E2 22373.093} C_VEL
LIN {X 0,Y 512.618,Z 409.2,A -85,B 0,C 180,E1 22372.023,E2 22372.023} C_VEL
LIN {X 0,Y 513.876,Z 374.612,A -85,B 0,C 180,E1 22371.49,E2 22371.49} C_VEL
LIN {X 0,Y 517.445,Z 358.291,A -85,B 0,C 180,E1 22370.847,E2 22370.847} C_VEL
LIN {X 0,Y 517.911,Z 317.946,A -85,B 0,C 180,E1 22368.071,E2 22368.071} C_VEL
LIN {X 0,Y 510.317,Z 297.328,A -85,B 0,C 180,E1 22365.614,E2 22365.614} C_VEL
LIN {X 0,Y 502.334,Z 278.601,A -85,B 0,C 180,E1 22363.215,E2 22363.215} C_VEL
LIN {X 0,Y 494.836,Z 263.053,A -85,B 0,C 180,E1 22361.05,E2 22361.05} C_VEL
LIN {X 0,Y 487.309,Z 249.107,A -85,B 0,C 180,E1 22358.954,E2 22358.954} C_VEL
LIN {X 0,Y 482.169,Z 240.332,A -85,B 0,C 180,E1 22357.566,E2 22357.566} C_VEL
LIN {X 0,Y 479.749,Z 236.125,A -85,B 0,C 180,E1 22356.888,E2 22356.888} C_VEL
LIN {X 0,Y 477.498,Z 232.436,A -85,B 0,C 180,E1 22356.274,E2 22356.274} C_VEL
LIN {X 0,Y 476.91,Z 231.296,A -85,B 0,C 180,E1 22356.097,E2 22356.097} C_VEL
LIN {X 0,Y 474.742,Z 228.427,A -85,B 0,C 180,E1 22355.543,E2 22355.543} C_VEL
LIN {X 0,Y 474.109,Z 226.17,A -85,B 0,C 180,E1 22355.258,E2 22355.258} C_VEL
LIN {X 0,Y 474.113,Z 226.159,A -85,B 0,C 180,E1 22351.536,E2 22351.536} C_VEL
LIN {X 0,Y 474.107,Z 226.143,A -85,B 0,C 180,E1 22347.912,E2 22347.912} C_VEL
LIN {X 0,Y 474.108,Z 226.139,A -85,B 0,C 180,E1 22344.284,E2 22344.284} C_VEL
LIN {X 0,Y 474.107,Z 226.173,A -85,B 0,C 180,E1 22340.622,E2 22340.622} C_VEL
LIN {X 0,Y 474.105,Z 226.141,A -85,B 0,C 180,E1 22336.92,E2 22336.92} C_VEL
LIN {X 0,Y 474.101,Z 226.141,A -85,B 0,C 180,E1 22333.415,E2 22333.415} C_VEL
LIN {X 0,Y 474.099,Z 226.17,A -85,B 0,C 180,E1 22329.714,E2 22329.714} C_VEL
